LIN {X 0,Y 230.991,Z 464.368,A -85,B 0,C 180,E1 -21092.538,E2 -21092.538} C_VEL
LIN {X 0,Y 229.288,Z 474.072,A -85,B 0,C 180,E1 -21093.412,E2 -21093.412} C_VEL
LIN {X 0,Y 227.158,Z 483.891,A -85,B 0,C 180,E1 -21094.538,E2 -21094.538} C_VEL
LIN {X 0,Y 224.562,Z 493.981,A -85,B 0,C 180,E1 -21096.008,E2 -21096.008} C_VEL
LIN {X 0,Y 221.905,Z 503.043,A -85,B 0,C 180,E1 -21097.648,E2 -21097.648} C_VEL
LIN {X 0,Y 218.983,Z 511.866,A -85,B 0,C 180,E1 -21099.624,E2 -21099.624} C_VEL
LIN {X 0,Y 216.287,Z 519.229,A -85,B 0,C 180,E1 -21101.638,E2 -21101.638} C_VEL
LIN {X 0,Y 213.888,Z 525.476,A -85,B 0,C 180,E1 -21103.707,E2 -21103.707} C_VEL
LIN {X 0,Y 211.783,Z 530.779,A -85,B 0,C 180,E1 -21105.823,E2 -21105.823} C_VEL
LIN {X 0,Y 209.103,Z 537.073,A -85,B 0,C 180,E1 -21109.05,E2 -21109.05} C_VEL
LIN {X 0,Y 207.83,Z 540.216,A -85,B 0,C 180,E1 -21111.057,E2 -21111.057} C_VEL
LIN {X 0,Y 205.854,Z 544.744,A -85,B 0,C 180,E1 -21115.023,E2 -21115.023} C_VEL
LIN {X 0,Y 205.221,Z 546.173,A -85,B 0,C 180,E1 -21116.775,E2 -21116.775} C_VEL
LIN {X 0,Y 204.564,Z 547.552,A -85,B 0,C 180,E1 -21119.194,E2 -21119.194} C_VEL
LIN {X 0,Y 204.178,Z 548.312,A -85,B 0,C 180,E1 -21121.191,E2 -21121.191} C_VEL
LIN {X 0,Y 203.917,Z 548.681,A -85,B 0,C 180,E1 -21123.65,E2 -21123.65} C_VEL
LIN {X 0,Y 203.84,Z 547.791,A -85,B 0,C 180,E1 -21127.712,E2 -21127.712} C_VEL
LIN {X 0,Y 204.07,Z 546.726,A -85,B 0,C 180,E1 -21129.855,E2 -21129.855} C_VEL
LIN {X 0,Y 204.801,Z 543.17,A -85,B 0,C 180,E1 -21133.917,E2 -21133.917} C_VEL
LIN {X 0,Y 205.395,Z 540.506,A -85,B 0,C 180,E1 -21136.142,E2 -21136.142} C_VEL
LIN {X 0,Y 206.522,Z 535.454,A -85,B 0,C 180,E1 -21139.312,E2 -21139.312} C_VEL
LIN {X 0,Y 208.013,Z 529.409,A -85,B 0,C 180,E1 -21142.233,E2 -21142.233} C_VEL
LIN {X 0,Y 209.693,Z 523.042,A -85,B 0,C 180,E1 -21144.712,E2 -21144.712} C_VEL
LIN {X 0,Y 211.428,Z 516.481,A -85,B 0,C 180,E1 -21146.829,E2 -21146.829} C_VEL
LIN {X 0,Y 213.706,Z 506.97,A -85,B 0,C 180,E1 -21149.294,E2 -21149.294} C_VEL
LIN {X 0,Y 215.821,Z 498.001,A -85,B 0,C 180,E1 -21151.166,E2 -21151.166} C_VEL
LIN {X 0,Y 217.545,Z 489.788,A -85,B 0,C 180,E1 -21152.594,E2 -21152.594} C_VEL
LIN {X 0,Y 219.548,Z 478.688,A -85,B 0,C 180,E1 -21154.131,E2 -21154.131} C_VEL
LIN {X 0,Y 221.149,Z 468.369,A -85,B 0,C 180,E1 -21155.242,E2 -21155.242} C_VEL
LIN {X 0,Y 222.36,Z 457.762,A -85,B 0,C 180,E1 -21156.124,E2 -21156.124} C_VEL
LIN {X 0,Y 223.449,Z 446.329,A -85,B 0,C 180,E1 -21156.774,E2 -21156.774} C_VEL
LIN {X 0,Y 224.548,Z 426.084,A -85,B 0,C 180,E1 -21157.478,E2 -21157.478} C_VEL
LIN {X 0,Y 226.379,Z 382.607,A -85,B 0,C 180,E1 -21158.855,E2 -21158.855} C_VEL
LIN {X 0,Y 221.699,Z 370.258,A -85,B 0,C 180,E1 -21159.987,E2 -21159.987} C_VEL
LIN {X 0,Y 215.137,Z 354.309,A -85,B 0,C 180,E1 -21161.622,E2 -21161.622} C_VEL
LIN {X 0,Y 208.262,Z 340.607,A -85,B 0,C 180,E1 -21163.351,E2 -21163.351} C_VEL
LIN {X 0,Y 207.018,Z 337.894,A -85,B 0,C 180,E1 -21163.81,E2 -21163.81} C_VEL
LIN {X 0,Y 206.912,Z 337.294,A -85,B 0,C 180,E1 -21164.256,E2 -21164.256} C_VEL
LIN {X 0,Y 206.86,Z 337.211,A -85,B 0,C 180,E1 -21167.956,E2 -21167.956} C_VEL
LIN {X 0,Y 206.756,Z 337.217,A -85,B 0,C 180,E1 -21173.396,E2 -21173.396} C_VEL
LIN {X 0,Y 206.739,Z 337.215,A -85,B 0,C 180,E1 -21178.42,E2 -21178.42} C_VEL
LIN {X 0,Y 206.708,Z 337.221,A -85,B 0,C 180,E1 -21182.956,E2 -21182.956} C_VEL
LIN {X 0,Y 206.724,Z 337.215,A -85,B 0,C 180,E1 -21185.32,E2 -21185.32} C_VEL
LIN {X 0,Y 206.669,Z 337.222,A -85,B 0,C 180,E1 -21190.25,E2 -21190.25} C_VEL
LIN {X 0,Y 206.637,Z 337.245,A -85,B 0,C 180,E1 -21195.581,E2 -21195.581} C_VEL
LIN {X 0,Y 206.663,Z 337.207,A -85,B 0,C 180,E1 -21199.749,E2 -21199.749} C_VEL
LIN {X 0,Y 206.701,Z 337.234,A -85,B 0,C 180,E1 -21204.689,E2 -21204.689} C_VEL
LIN {X 0,Y 206.697,Z 337.198,A -85,B 0,C 180,E1 -21209.334,E2 -21209.334} C_VEL
LIN {X 0,Y 206.709,Z 337.222,A -85,B 0,C 180,E1 -21213.768,E2 -21213.768} C_VEL
LIN {X 0,Y 206.737,Z 337.222,A -85,B 0,C 180,E1 -21218.04,E2 -21218.04} C_VEL
LIN {X 0,Y 206.828,Z 337.17,A -85,B 0,C 180,E1 -21222.192,E2 -21222.192} C_VEL
LIN {X 0,Y 206.884,Z 337.209,A -85,B 0,C 180,E1 -21226.243,E2 -21226.243} C_VEL
LIN {X 0,Y 207.08,Z 337.176,A -85,B 0,C 180,E1 -21230.23,E2 -21230.23} C_VEL
LIN {X 0,Y 207.04,Z 337.145,A -85,B 0,C 180,E1 -21234.155,E2 -21234.155} C_VEL
LIN {X 0,Y 207.347,Z 337.149,A -85,B 0,C 180,E1 -21238.057,E2 -21238.057} C_VEL
LIN {X 0,Y 207.484,Z 337.138,A -85,B 0,C 180,E1 -21240,E2 -21240} C_VEL
LIN {X 0,Y 207.348,Z 337.138,A -85,B 0,C 180,E1 -21241.942,E2 -21241.942} C_VEL
LIN {X 0,Y 207.134,Z 337.166,A -85,B 0,C 180,E1 -21247.8,E2 -21247.8} C_VEL
LIN {X 0,Y 207.063,Z 337.192,A -85,B 0,C 180,E1 -21250.164,E2 -21250.164} C_VEL
LIN {X 0,Y 206.801,Z 337.189,A -85,B 0,C 180,E1 -21255.775,E2 -21255.775} C_VEL
LIN {X 0,Y 206.714,Z 337.237,A -85,B 0,C 180,E1 -21259.875,E2 -21259.875} C_VEL
LIN {X 0,Y 206.735,Z 337.204,A -85,B 0,C 180,E1 -21264.075,E2 -21264.075} C_VEL
LIN {X 0,Y 206.689,Z 337.238,A -85,B 0,C 180,E1 -21268.426,E2 -21268.426} C_VEL
LIN {X 0,Y 206.694,Z 337.228,A -85,B 0,C 180,E1 -21272.958,E2 -21272.958} C_VEL
LIN {X 0,Y 206.699,Z 337.235,A -85,B 0,C 180,E1 -21275.311,E2 -21275.311} C_VEL
LIN {X 0,Y 206.643,Z 337.245,A -85,B 0,C 180,E1 -21280.255,E2 -21280.255} C_VEL
LIN {X 0,Y 206.622,Z 337.243,A -85,B 0,C 180,E1 -21285.355,E2 -21285.355} C_VEL
LIN {X 0,Y 206.702,Z 337.357,A -85,B 0,C 180,E1 -21289.626,E2 -21289.626} C_VEL
LIN {X 0,Y 207.203,Z 339.383,A -85,B 0,C 180,E1 -21290.808,E2 -21290.808} C_VEL
LIN {X 0,Y 207.694,Z 341.656,A -85,B 0,C 180,E1 -21291.645,E2 -21291.645} C_VEL
LIN {X 0,Y 208.362,Z 345.527,A -85,B 0,C 180,E1 -21292.422,E2 -21292.422} C_VEL
LIN {X 0,Y 209.256,Z 351.887,A -85,B 0,C 180,E1 -21293.126,E2 -21293.126} C_VEL
LIN {X 0,Y 211.154,Z 364.004,A -85,B 0,C 180,E1 -21293.947,E2 -21293.947} C_VEL
LIN {X 0,Y 212.237,Z 367.853,A -85,B 0,C 180,E1 -21294.286,E2 -21294.286} C_VEL
LIN {X 0,Y 218.175,Z 383.461,A -85,B 0,C 180,E1 -21295.828,E2 -21295.828} C_VEL
LIN {X 0,Y 219.745,Z 395.439,A -85,B 0,C 180,E1 -21296.523,E2 -21296.523} C_VEL
LIN {X 0,Y 217.151,Z 449.684,A -85,B 0,C 180,E1 -21298.324,E2 -21298.324} C_VEL
LIN {X 0,Y 216.405,Z 459.263,A -85,B 0,C 180,E1 -21298.829,E2 -21298.829} C_VEL
LIN {X 0,Y 215.141,Z 469.584,A -85,B 0,C 180,E1 -21299.579,E2 -21299.579} C_VEL
LIN {X 0,Y 213.699,Z 478.713,A -85,B 0,C 180,E1 -21300.441,E2 -21300.441} C_VEL
LIN {X 0,Y 211.865,Z 489.444,A -85,B 0,C 180,E1 -21301.79,E2 -21301.79} C_VEL
LIN {X 0,Y 209.66,Z 499.462,A -85,B 0,C 180,E1 -21303.362,E2 -21303.362} C_VEL
LIN {X 0,Y 207.477,Z 508.858,A -85,B 0,C 180,E1 -21305.217,E2 -21305.217} C_VEL
LIN {X 0,Y 205.84,Z 515.883,A -85,B 0,C 180,E1 -21306.881,E2 -21306.881} C_VEL
LIN {X 0,Y 203.685,Z 524.444,A -85,B 0,C 180,E1 -21309.374,E2 -21309.374} C_VEL
LIN {X 0,Y 201.845,Z 531.126,A -85,B 0,C 180,E1 -21311.737,E2 -21311.737} C_VEL
LIN {X 0,Y 200.242,Z 536.899,A -85,B 0,C 180,E1 -21314.216,E2 -21314.216} C_VEL
LIN {X 0,Y 199.057,Z 541.697,A -85,B 0,C 180,E1 -21316.733,E2 -21316.733} C_VEL
LIN {X 0,Y 198.081,Z 546.272,A -85,B 0,C 180,E1 -21319.781,E2 -21319.781} C_VEL
LIN {X 0,Y 197.345,Z 550.566,A -85,B 0,C 180,E1 -21323.867,E2 -21323.867} C_VEL
LIN {X 0,Y 197.144,Z 552.501,A -85,B 0,C 180,E1 -21326.525,E2 -21326.525} C_VEL
LIN {X 0,Y 197.242,Z 553.89,A -85,B 0,C 180,E1 -21330,E2 -21330} C_VEL
LIN {X 0,Y 197.19,Z 554.197,A -85,B 0,C 180,E1 -21332.042,E2 -21332.042} C_VEL
LIN {X 0,Y 197.408,Z 553.575,A -85,B 0,C 180,E1 -21336.131,E2 -21336.131} C_VEL
LIN {X 0,Y 198.182,Z 551.263,A -85,B 0,C 180,E1 -21340.213,E2 -21340.213} C_VEL
LIN {X 0,Y 199.305,Z 548.5,A -85,B 0,C 180,E1 -21343.25,E2 -21343.25} C_VEL
LIN {X 0,Y 200.827,Z 544.728,A -85,B 0,C 180,E1 -21346.258,E2 -21346.258} C_VEL
LIN {X 0,Y 203.105,Z 539.836,A -85,B 0,C 180,E1 -21349.191,E2 -21349.191} C_VEL
LIN {X 0,Y 205.282,Z 534.853,A -85,B 0,C 180,E1 -21351.594,E2 -21351.594} C_VEL
LIN {X 0,Y 208.16,Z 527.463,A -85,B 0,C 180,E1 -21354.43,E2 -21354.43} C_VEL
LIN {X 0,Y 211.104,Z 519.997,A -85,B 0,C 180,E1 -21356.707,E2 -21356.707} C_VEL
LIN {X 0,Y 213.733,Z 512.974,A -85,B 0,C 180,E1 -21358.476,E2 -21358.476} C_VEL
LIN {X 0,Y 216.843,Z 503.458,A -85,B 0,C 180,E1 -21360.425,E2 -21360.425} C_VEL
LIN {X 0,Y 219.6,Z 494.547,A -85,B 0,C 180,E1 -21361.874,E2 -21361.874} C_VEL
LIN {X 0,Y 221.939,Z 485.384,A -85,B 0,C 180,E1 -21363.11,E2 -21363.11} C_VEL
LIN {X 0,Y 224.415,Z 473.711,A -85,B 0,C 180,E1 -21364.312,E2 -21364.312} C_VEL
LIN {X 0,Y 226.285,Z 462.828,A -85,B 0,C 180,E1 -21365.138,E2 -21365.138} C_VEL
LIN {X 0,Y 227.665,Z 452.178,A -85,B 0,C 180,E1 -21365.706,E2 -21365.706} C_VEL
LIN {X 0,Y 228.836,Z 433.635,A -85,B 0,C 180,E1 -21366.376,E2 -21366.376} C_VEL
LIN {X 0,Y 230.861,Z 397.556,A -85,B 0,C 180,E1 -21367.506,E2 -21367.506} C_VEL
LIN {X 0,Y 230.289,Z 394.728,A -85,B 0,C 180,E1 -21367.764,E2 -21367.764} C_VEL
LIN {X 0,Y 225.862,Z 383.934,A -85,B 0,C 180,E1 -21369.337,E2 -21369.337} C_VEL
LIN {X 0,Y 221.04,Z 373.739,A -85,B 0,C 180,E1 -21371.113,E2 -21371.113} C_VEL
LIN {X 0,Y 215.575,Z 363.857,A -85,B 0,C 180,E1 -21373.241,E2 -21373.241} C_VEL
LIN {X 0,Y 211.072,Z 356.624,A -85,B 0,C 180,E1 -21375.117,E2 -21375.117} C_VEL
LIN {X 0,Y 207.674,Z 351.407,A -85,B 0,C 180,E1 -21376.652,E2 -21376.652} C_VEL
LIN {X 0,Y 203.916,Z 345.962,A -85,B 0,C 180,E1 -21378.495,E2 -21378.495} C_VEL
LIN {X 0,Y 200.8,Z 341.569,A -85,B 0,C 180,E1 -21380.188,E2 -21380.188} C_VEL
LIN {X 0,Y 200.327,Z 340.412,A -85,B 0,C 180,E1 -21380.841,E2 -21380.841} C_VEL
LIN {X 0,Y 199.603,Z 338.146,A -85,B 0,C 180,E1 -21383.076,E2 -21383.076} C_VEL
LIN {X 0,Y 199.693,Z 338.1,A -85,B 0,C 180,E1 -21388.136,E2 -21388.136} C_VEL
LIN {X 0,Y 199.686,Z 338.099,A -85,B 0,C 180,E1 -21392.772,E2 -21392.772} C_VEL
LIN {X 0,Y 199.738,Z 338.091,A -85,B 0,C 180,E1 -21397.23,E2 -21397.23} C_VEL
LIN {X 0,Y 199.797,Z 338.082,A -85,B 0,C 180,E1 -21401.758,E2 -21401.758} C_VEL
LIN {X 0,Y 199.849,Z 338.076,A -85,B 0,C 180,E1 -21405.75,E2 -21405.75} C_VEL
LIN {X 0,Y 200.076,Z 338.052,A -85,B 0,C 180,E1 -21409.885,E2 -21409.885} C_VEL
LIN {X 0,Y 200.039,Z 338.065,A -85,B 0,C 180,E1 -21413.95,E2 -21413.95} C_VEL
LIN {X 0,Y 200.324,Z 338.032,A -85,B 0,C 180,E1 -21417.99,E2 -21417.99} C_VEL
LIN {X 0,Y 200.481,Z 337.999,A -85,B 0,C 180,E1 -21420,E2 -21420} C_VEL
LIN {X 0,Y 200.034,Z 338.057,A -85,B 0,C 180,E1 -21424.03,E2 -21424.03} C_VEL
LIN {X 0,Y 200.134,Z 338.047,A -85,B 0,C 180,E1 -21428.075,E2 -21428.075} C_VEL
LIN {X 0,Y 199.889,Z 338.077,A -85,B 0,C 180,E1 -21432.179,E2 -21432.179} C_VEL
LIN {X 0,Y 199.833,Z 338.258,A -85,B 0,C 180,E1 -21435.36,E2 -21435.36} C_VEL
LIN {X 0,Y 201.002,Z 341.243,A -85,B 0,C 180,E1 -21436.179,E2 -21436.179} C_VEL
LIN {X 0,Y 203.144,Z 343.29,A -85,B 0,C 180,E1 -21437.253,E2 -21437.253} C_VEL
LIN {X 0,Y 203.866,Z 343.978,A -85,B 0,C 180,E1 -21437.603,E2 -21437.603} C_VEL
LIN {X 0,Y 205.814,Z 347.16,A -85,B 0,C 180,E1 -21438.607,E2 -21438.607} C_VEL
LIN {X 0,Y 207.679,Z 349.151,A -85,B 0,C 180,E1 -21439.459,E2 -21439.459} C_VEL
LIN {X 0,Y 211.882,Z 355.373,A -85,B 0,C 180,E1 -21441.336,E2 -21441.336} C_VEL
LIN {X 0,Y 216.905,Z 363.24,A -85,B 0,C 180,E1 -21443.386,E2 -21443.386} C_VEL
LIN {X 0,Y 223.704,Z 375.723,A -85,B 0,C 180,E1 -21445.955,E2 -21445.955} C_VEL
LIN {X 0,Y 228.725,Z 386.551,A -85,B 0,C 180,E1 -21447.746,E2 -21447.746} C_VEL
LIN {X 0,Y 231.231,Z 393.178,A -85,B 0,C 180,E1 -21448.632,E2 -21448.632} C_VEL
LIN {X 0,Y 228.008,Z 444.485,A -85,B 0,C 180,E1 -21450.237,E2 -21450.237} C_VEL
LIN {X 0,Y 226.966,Z 454.3,A -85,B 0,C 180,E1 -21450.71,E2 -21450.71} C_VEL
LIN {X 0,Y 225.472,Z 464.664,A -85,B 0,C 180,E1 -21451.429,E2 -21451.429} C_VEL
LIN {X 0,Y 223.773,Z 473.933,A -85,B 0,C 180,E1 -21452.271,E2 -21452.271} C_VEL
LIN {X 0,Y 221.315,Z 484.658,A -85,B 0,C 180,E1 -21453.531,E2 -21453.531} C_VEL
LIN {X 0,Y 218.917,Z 493.605,A -85,B 0,C 180,E1 -21454.849,E2 -21454.849} C_VEL
LIN {X 0,Y 215.848,Z 503.572,A -85,B 0,C 180,E1 -21456.699,E2 -21456.699} C_VEL
LIN {X 0,Y 213.037,Z 511.63,A -85,B 0,C 180,E1 -21458.535,E2 -21458.535} C_VEL
LIN {X 0,Y 210.307,Z 518.789,A -85,B 0,C 180,E1 -21460.514,E2 -21460.514} C_VEL
LIN {X 0,Y 207.111,Z 526.53,A -85,B 0,C 180,E1 -21463.194,E2 -21463.194} C_VEL
LIN {X 0,Y 204.962,Z 531.617,A -85,B 0,C 180,E1 -21465.339,E2 -21465.339} C_VEL
LIN {X 0,Y 203.064,Z 535.949,A -85,B 0,C 180,E1 -21467.555,E2 -21467.555} C_VEL
LIN {X 0,Y 200.741,Z 541.076,A -85,B 0,C 180,E1 -21470.936,E2 -21470.936} C_VEL
LIN {X 0,Y 198.994,Z 544.736,A -85,B 0,C 180,E1 -21474.322,E2 -21474.322} C_VEL
LIN {X 0,Y 197.585,Z 547.577,A -85,B 0,C 180,E1 -21478.614,E2 -21478.614} C_VEL
LIN {X 0,Y 197.275,Z 548.247,A -85,B 0,C 180,E1 -21480.083,E2 -21480.083} C_VEL
LIN {X 0,Y 196.838,Z 548.764,A -85,B 0,C 180,E1 -21483.204,E2 -21483.204} C_VEL
LIN {X 0,Y 196.711,Z 548.233,A -85,B 0,C 180,E1 -21486.859,E2 -21486.859} C_VEL
LIN {X 0,Y 196.862,Z 547.189,A -85,B 0,C 180,E1 -21489.084,E2 -21489.084} C_VEL
LIN {X 0,Y 197.159,Z 545.745,A -85,B 0,C 180,E1 -21491.288,E2 -21491.288} C_VEL
LIN {X 0,Y 197.656,Z 543.611,A -85,B 0,C 180,E1 -21493.747,E2 -21493.747} C_VEL
LIN {X 0,Y 198.437,Z 540.125,A -85,B 0,C 180,E1 -21496.691,E2 -21496.691} C_VEL
LIN {X 0,Y 199.753,Z 534.627,A -85,B 0,C 180,E1 -21500.111,E2 -21500.111} C_VEL
LIN {X 0,Y 201.304,Z 528.712,A -85,B 0,C 180,E1 -21502.981,E2 -21502.981} C_VEL
LIN {X 0,Y 203.073,Z 522.187,A -85,B 0,C 180,E1 -21505.534,E2 -21505.534} C_VEL
LIN {X 0,Y 205.192,Z 514.275,A -85,B 0,C 180,E1 -21508.037,E2 -21508.037} C_VEL
LIN {X 0,Y 207.068,Z 506.764,A -85,B 0,C 180,E1 -21510,E2 -21510} C_VEL
LIN {X 0,Y 209.299,Z 497.72,A -85,B 0,C 180,E1 -21511.924,E2 -21511.924} C_VEL
LIN {X 0,Y 211.234,Z 488.729,A -85,B 0,C 180,E1 -21513.494,E2 -21513.494} C_VEL
LIN {X 0,Y 212.863,Z 480.134,A -85,B 0,C 180,E1 -21514.735,E2 -21514.735} C_VEL
LIN {X 0,Y 214.691,Z 468.951,A -85,B 0,C 180,E1 -21515.99,E2 -21515.99} C_VEL
LIN {X 0,Y 215.997,Z 457.719,A -85,B 0,C 180,E1 -21516.95,E2 -21516.95} C_VEL
LIN {X 0,Y 217.092,Z 447.007,A -85,B 0,C 180,E1 -21517.578,E2 -21517.578} C_VEL
LIN {X 0,Y 218.099,Z 429.281,A -85,B 0,C 180,E1 -21518.229,E2 -21518.229} C_VEL
LIN {X 0,Y 220.105,Z 384.246,A -85,B 0,C 180,E1 -21519.686,E2 -21519.686} C_VEL
LIN {X 0,Y 215.374,Z 371.866,A -85,B 0,C 180,E1 -21520.883,E2 -21520.883} C_VEL
LIN {X 0,Y 209.688,Z 357.873,A -85,B 0,C 180,E1 -21522.375,E2 -21522.375} C_VEL
LIN {X 0,Y 202.814,Z 344.277,A -85,B 0,C 180,E1 -21524.162,E2 -21524.162} C_VEL
LIN {X 0,Y 200.134,Z 339.336,A -85,B 0,C 180,E1 -21524.912,E2 -21524.912} C_VEL
LIN {X 0,Y 199.868,Z 338.298,A -85,B 0,C 180,E1 -21525.29,E2 -21525.29} C_VEL
LIN {X 0,Y 199.783,Z 338.09,A -85,B 0,C 180,E1 -21528.458,E2 -21528.458} C_VEL
LIN {X 0,Y 199.717,Z 338.095,A -85,B 0,C 180,E1 -21533.803,E2 -21533.803} C_VEL
LIN {X 0,Y 199.71,Z 338.09,A -85,B 0,C 180,E1 -21538.384,E2 -21538.384} C_VEL
LIN {X 0,Y 199.66,Z 338.107,A -85,B 0,C 180,E1 -21542.349,E2 -21542.349} C_VEL
LIN {X 0,Y 199.642,Z 338.113,A -85,B 0,C 180,E1 -21546.759,E2 -21546.759} C_VEL
LIN {X 0,Y 199.641,Z 338.108,A -85,B 0,C 180,E1 -21549.321,E2 -21549.321} C_VEL
LIN {X 0,Y 199.584,Z 338.12,A -85,B 0,C 180,E1 -21554.77,E2 -21554.77} C_VEL
LIN {X 0,Y 199.582,Z 338.107,A -85,B 0,C 180,E1 -21558.005,E2 -21558.005} C_VEL
LIN {X 0,Y 199.612,Z 338.082,A -85,B 0,C 180,E1 -21560.768,E2 -21560.768} C_VEL
LIN {X 0,Y 199.613,Z 338.119,A -85,B 0,C 180,E1 -21565.713,E2 -21565.713} C_VEL
LIN {X 0,Y 199.688,Z 338.087,A -85,B 0,C 180,E1 -21568.134,E2 -21568.134} C_VEL
LIN {X 0,Y 199.646,Z 338.086,A -85,B 0,C 180,E1 -21572.765,E2 -21572.765} C_VEL
LIN {X 0,Y 199.711,Z 338.104,A -85,B 0,C 180,E1 -21577.225,E2 -21577.225} C_VEL
LIN {X 0,Y 199.752,Z 338.05,A -85,B 0,C 180,E1 -21581.798,E2 -21581.798} C_VEL
LIN {X 0,Y 199.821,Z 338.082,A -85,B 0,C 180,E1 -21585.747,E2 -21585.747} C_VEL
LIN {X 0,Y 200.025,Z 338.056,A -85,B 0,C 180,E1 -21589.881,E2 -21589.881} C_VEL
LIN {X 0,Y 200.004,Z 338.02,A -85,B 0,C 180,E1 -21593.948,E2 -21593.948} C_VEL
LIN {X 0,Y 200.289,Z 338.028,A -85,B 0,C 180,E1 -21597.989,E2 -21597.989} C_VEL
LIN {X 0,Y 200.451,Z 338.014,A -85,B 0,C 180,E1 -21600,E2 -21600} C_VEL
LIN {X 0,Y 199.993,Z 338.029,A -85,B 0,C 180,E1 -21604.03,E2 -21604.03} C_VEL
LIN {X 0,Y 200.084,Z 338.048,A -85,B 0,C 180,E1 -21608.076,E2 -21608.076} C_VEL
LIN {X 0,Y 199.857,Z 338.08,A -85,B 0,C 180,E1 -21612.18,E2 -21612.18} C_VEL
LIN {X 0,Y 199.742,Z 338.072,A -85,B 0,C 180,E1 -21616.348,E2 -21616.348} C_VEL
LIN {X 0,Y 199.647,Z 338.113,A -85,B 0,C 180,E1 -21620.61,E2 -21620.61} C_VEL
LIN {X 0,Y 199.649,Z 338.09,A -85,B 0,C 180,E1 -21624.987,E2 -21624.987} C_VEL
LIN {X 0,Y 199.609,Z 338.109,A -85,B 0,C 180,E1 -21629.532,E2 -21629.532} C_VEL
LIN {X 0,Y 199.665,Z 338.096,A -85,B 0,C 180,E1 -21632.352,E2 -21632.352} C_VEL
LIN {X 0,Y 199.614,Z 338.104,A -85,B 0,C 180,E1 -21636.764,E2 -21636.764} C_VEL
LIN {X 0,Y 199.592,Z 338.12,A -85,B 0,C 180,E1 -21639.331,E2 -21639.331} C_VEL
LIN {X 0,Y 199.563,Z 338.113,A -85,B 0,C 180,E1 -21642.306,E2 -21642.306} C_VEL
LIN {X 0,Y 199.575,Z 338.123,A -85,B 0,C 180,E1 -21645.227,E2 -21645.227} C_VEL
LIN {X 0,Y 199.654,Z 338.34,A -85,B 0,C 180,E1 -21648.805,E2 -21648.805} C_VEL
LIN {X 0,Y 200.775,Z 342.66,A -85,B 0,C 180,E1 -21651.153,E2 -21651.153} C_VEL
LIN {X 0,Y 206.804,Z 355.302,A -85,B 0,C 180,E1 -21652.852,E2 -21652.852} C_VEL
LIN {X 0,Y 212.237,Z 367.853,A -85,B 0,C 180,E1 -21654.286,E2 -21654.286} C_VEL
LIN {X 0,Y 213.639,Z 373.386,A -85,B 0,C 180,E1 -21654.735,E2 -21654.735} C_VEL
LIN {X 0,Y 214.2,Z 379.209,A -85,B 0,C 180,E1 -21655.058,E2 -21655.058} C_VEL
LIN {X 0,Y 213.825,Z 391.21,A -85,B 0,C 180,E1 -21655.485,E2 -21655.485} C_VEL
LIN {X 0,Y 213.327,Z 399.271,A -85,B 0,C 180,E1 -21655.734,E2 -21655.734} C_VEL
LIN {X 0,Y 210.886,Z 449.057,A -85,B 0,C 180,E1 -21657.431,E2 -21657.431} C_VEL
LIN {X 0,Y 210.138,Z 458.563,A -85,B 0,C 180,E1 -21657.931,E2 -21657.931} C_VEL
LIN {X 0,Y 208.851,Z 469.048,A -85,B 0,C 180,E1 -21658.702,E2 -21658.702} C_VEL
LIN {X 0,Y 207.18,Z 479.208,A -85,B 0,C 180,E1 -21659.695,E2 -21659.695} C_VEL
LIN {X 0,Y 205.275,Z 489.825,A -85,B 0,C 180,E1 -21661.079,E2 -21661.079} C_VEL
LIN {X 0,Y 202.989,Z 499.756,A -85,B 0,C 180,E1 -21662.693,E2 -21662.693} C_VEL
LIN {X 0,Y 201.004,Z 508.057,A -85,B 0,C 180,E1 -21664.362,E2 -21664.362} C_VEL
LIN {X 0,Y 198.806,Z 516.925,A -85,B 0,C 180,E1 -21666.565,E2 -21666.565} C_VEL
LIN {X 0,Y 196.947,Z 524.021,A -85,B 0,C 180,E1 -21668.695,E2 -21668.695} C_VEL
LIN {X 0,Y 195.046,Z 530.628,A -85,B 0,C 180,E1 -21671.077,E2 -21671.077} C_VEL
LIN {X 0,Y 193.081,Z 537.444,A -85,B 0,C 180,E1 -21674.157,E2 -21674.157} C_VEL
LIN {X 0,Y 191.715,Z 542.899,A -85,B 0,C 180,E1 -21677.294,E2 -21677.294} C_VEL
LIN {X 0,Y 191.07,Z 545.952,A -85,B 0,C 180,E1 -21679.402,E2 -21679.402} C_VEL
LIN {X 0,Y 190.424,Z 549.47,A -85,B 0,C 180,E1 -21682.578,E2 -21682.578} C_VEL
LIN {X 0,Y 190.087,Z 551.956,A -85,B 0,C 180,E1 -21685.759,E2 -21685.759} C_VEL
LIN {X 0,Y 190.15,Z 553.763,A -85,B 0,C 180,E1 -21690,E2 -21690} C_VEL
LIN {X 0,Y 190.092,Z 554.066,A -85,B 0,C 180,E1 -21693.418,E2 -21693.418} C_VEL
LIN {X 0,Y 190.352,Z 553.546,A -85,B 0,C 180,E1 -21696.359,E2 -21696.359} C_VEL
LIN {X 0,Y 191.17,Z 551.297,A -85,B 0,C 180,E1 -21700.592,E2 -21700.592} C_VEL
LIN {X 0,Y 192.375,Z 548.591,A -85,B 0,C 180,E1 -21703.737,E2 -21703.737} C_VEL
LIN {X 0,Y 194.008,Z 544.878,A -85,B 0,C 180,E1 -21706.846,E2 -21706.846} C_VEL
LIN {X 0,Y 196.412,Z 540.061,A -85,B 0,C 180,E1 -21709.872,E2 -21709.872} C_VEL
LIN {X 0,Y 198.689,Z 535.165,A -85,B 0,C 180,E1 -21712.349,E2 -21712.349} C_VEL
LIN {X 0,Y 201.727,Z 527.881,A -85,B 0,C 180,E1 -21715.263,E2 -21715.263} C_VEL
LIN {X 0,Y 204.818,Z 520.519,A -85,B 0,C 180,E1 -21717.596,E2 -21717.596} C_VEL
LIN {X 0,Y 207.895,Z 512.607,A -85,B 0,C 180,E1 -21719.63,E2 -21719.63} C_VEL
LIN {X 0,Y 211.209,Z 503.03,A -85,B 0,C 180,E1 -21721.606,E2 -21721.606} C_VEL
LIN {X 0,Y 214.065,Z 494.05,A -85,B 0,C 180,E1 -21723.08,E2 -21723.08} C_VEL
LIN {X 0,Y 216.521,Z 484.788,A -85,B 0,C 180,E1 -21724.331,E2 -21724.331} C_VEL
LIN {X 0,Y 218.881,Z 474.157,A -85,B 0,C 180,E1 -21725.448,E2 -21725.448} C_VEL
LIN {X 0,Y 220.931,Z 462.669,A -85,B 0,C 180,E1 -21726.333,E2 -21726.333} C_VEL
LIN {X 0,Y 222.353,Z 452.001,A -85,B 0,C 180,E1 -21726.908,E2 -21726.908} C_VEL
LIN {X 0,Y 223.571,Z 433.989,A -85,B 0,C 180,E1 -21727.57,E2 -21727.57} C_VEL
LIN {X 0,Y 225.662,Z 398.776,A -85,B 0,C 180,E1 -21728.691,E2 -21728.691} C_VEL
LIN {X 0,Y 221.567,Z 388.303,A -85,B 0,C 180,E1 -21730.249,E2 -21730.249} C_VEL
LIN {X 0,Y 216.908,Z 378.241,A -85,B 0,C 180,E1 -21732.067,E2 -21732.067} C_VEL
LIN {X 0,Y 211.283,Z 367.762,A -85,B 0,C 180,E1 -21734.412,E2 -21734.412} C_VEL
LIN {X 0,Y 204.983,Z 357.55,A -85,B 0,C 180,E1 -21737.301,E2 -21737.301} C_VEL
LIN {X 0,Y 200.852,Z 351.538,A -85,B 0,C 180,E1 -21739.413,E2 -21739.413} C_VEL
LIN {X 0,Y 196.941,Z 346.172,A -85,B 0,C 180,E1 -21741.599,E2 -21741.599} C_VEL
LIN {X 0,Y 193.033,Z 340.765,A -85,B 0,C 180,E1 -21744.244,E2 -21744.244} C_VEL
LIN {X 0,Y 192.572,Z 339.065,A -85,B 0,C 180,E1 -21746.025,E2 -21746.025} C_VEL
LIN {X 0,Y 192.648,Z 338.984,A -85,B 0,C 180,E1 -21751.109,E2 -21751.109} C_VEL
LIN {X 0,Y 192.706,Z 338.968,A -85,B 0,C 180,E1 -21756.349,E2 -21756.349} C_VEL
LIN {X 0,Y 192.732,Z 338.962,A -85,B 0,C 180,E1 -21761.458,E2 -21761.458} C_VEL
LIN {X 0,Y 192.773,Z 338.96,A -85,B 0,C 180,E1 -21765.215,E2 -21765.215} C_VEL
LIN {X 0,Y 193.021,Z 338.934,A -85,B 0,C 180,E1 -21769.511,E2 -21769.511} C_VEL
LIN {X 0,Y 193.003,Z 338.944,A -85,B 0,C 180,E1 -21773.729,E2 -21773.729} C_VEL
LIN {X 0,Y 193.266,Z 338.91,A -85,B 0,C 180,E1 -21777.917,E2 -21777.917} C_VEL
LIN {X 0,Y 193.445,Z 338.875,A -85,B 0,C 180,E1 -21780.001,E2 -21780.001} C_VEL
LIN {X 0,Y 192.981,Z 338.935,A -85,B 0,C 180,E1 -21784.177,E2 -21784.177} C_VEL
LIN {X 0,Y 193.081,Z 338.924,A -85,B 0,C 180,E1 -21788.372,E2 -21788.372} C_VEL
LIN {X 0,Y 192.9,Z 339.125,A -85,B 0,C 180,E1 -21791.893,E2 -21791.893} C_VEL
LIN {X 0,Y 193.757,Z 341.715,A -85,B 0,C 180,E1 -21792.63,E2 -21792.63} C_VEL
LIN {X 0,Y 195.632,Z 343.816,A -85,B 0,C 180,E1 -21793.82,E2 -21793.82} C_VEL
LIN {X 0,Y 197.126,Z 344.902,A -85,B 0,C 180,E1 -21794.65,E2 -21794.65} C_VEL
LIN {X 0,Y 198.873,Z 347.938,A -85,B 0,C 180,E1 -21795.698,E2 -21795.698} C_VEL
LIN {X 0,Y 201.182,Z 350.339,A -85,B 0,C 180,E1 -21796.899,E2 -21796.899} C_VEL
LIN {X 0,Y 203.625,Z 353.786,A -85,B 0,C 180,E1 -21798.163,E2 -21798.163} C_VEL
LIN {X 0,Y 204.977,Z 355.5,A -85,B 0,C 180,E1 -21798.815,E2 -21798.815} C_VEL
LIN {X 0,Y 208.64,Z 361.017,A -85,B 0,C 180,E1 -21800.535,E2 -21800.535} C_VEL
LIN {X 0,Y 213.19,Z 368.292,A -85,B 0,C 180,E1 -21802.492,E2 -21802.492} C_VEL
LIN {X 0,Y 219.634,Z 380.477,A -85,B 0,C 180,E1 -21805.082,E2 -21805.082} C_VEL
LIN {X 0,Y 224.103,Z 390.285,A -85,B 0,C 180,E1 -21806.76,E2 -21806.76} C_VEL
LIN {X 0,Y 225.941,Z 394.893,A -85,B 0,C 180,E1 -21807.444,E2 -21807.444} C_VEL
LIN {X 0,Y 222.727,Z 444.505,A -85,B 0,C 180,E1 -21809.035,E2 -21809.035} C_VEL
LIN {X 0,Y 221.608,Z 454.525,A -85,B 0,C 180,E1 -21809.525,E2 -21809.525} C_VEL
LIN {X 0,Y 220.111,Z 464.484,A -85,B 0,C 180,E1 -21810.221,E2 -21810.221} C_VEL
LIN {X 0,Y 218.19,Z 474.493,A -85,B 0,C 180,E1 -21811.15,E2 -21811.15} C_VEL
LIN {X 0,Y 216.042,Z 483.76,A -85,B 0,C 180,E1 -21812.243,E2 -21812.243} C_VEL
LIN {X 0,Y 213.264,Z 493.557,A -85,B 0,C 180,E1 -21813.685,E2 -21813.685} C_VEL
LIN {X 0,Y 210.267,Z 502.966,A -85,B 0,C 180,E1 -21815.441,E2 -21815.441} C_VEL
LIN {X 0,Y 207.012,Z 511.856,A -85,B 0,C 180,E1 -21817.5,E2 -21817.5} C_VEL
LIN {X 0,Y 203.695,Z 519.999,A -85,B 0,C 180,E1 -21819.854,E2 -21819.854} C_VEL
LIN {X 0,Y 201.062,Z 526.116,A -85,B 0,C 180,E1 -21822.021,E2 -21822.021} C_VEL
LIN {X 0,Y 198.165,Z 532.449,A -85,B 0,C 180,E1 -21824.822,E2 -21824.822} C_VEL
LIN {X 0,Y 196.185,Z 536.692,A -85,B 0,C 180,E1 -21827.106,E2 -21827.106} C_VEL
LIN {X 0,Y 193.758,Z 541.601,A -85,B 0,C 180,E1 -21830.598,E2 -21830.598} C_VEL
LIN {X 0,Y 191.931,Z 545.158,A -85,B 0,C 180,E1 -21834.135,E2 -21834.135} C_VEL
LIN {X 0,Y 191.076,Z 546.927,A -85,B 0,C 180,E1 -21836.515,E2 -21836.515} C_VEL
LIN {X 0,Y 190.419,Z 548.003,A -85,B 0,C 180,E1 -21838.888,E2 -21838.888} C_VEL
LIN {X 0,Y 189.793,Z 548.835,A -85,B 0,C 180,E1 -21842.713,E2 -21842.713} C_VEL
LIN {X 0,Y 189.614,Z 548.487,A -85,B 0,C 180,E1 -21845.939,E2 -21845.939} C_VEL
LIN {X 0,Y 189.705,Z 547.642,A -85,B 0,C 180,E1 -21848.256,E2 -21848.256} C_VEL
LIN {X 0,Y 189.921,Z 546.432,A -85,B 0,C 180,E1 -21850.547,E2 -21850.547} C_VEL
LIN {X 0,Y 190.508,Z 544.021,A -85,B 0,C 180,E1 -21853.571,E2 -21853.571} C_VEL
LIN {X 0,Y 191.518,Z 539.678,A -85,B 0,C 180,E1 -21857.281,E2 -21857.281} C_VEL
LIN {X 0,Y 192.607,Z 535.318,A -85,B 0,C 180,E1 -21860.132,E2 -21860.132} C_VEL
LIN {X 0,Y 194.274,Z 529.208,A -85,B 0,C 180,E1 -21863.248,E2 -21863.248} C_VEL
LIN {X 0,Y 196.105,Z 522.76,A -85,B 0,C 180,E1 -21865.89,E2 -21865.89} C_VEL
LIN {X 0,Y 197.855,Z 516.708,A -85,B 0,C 180,E1 -21867.965,E2 -21867.965} C_VEL
LIN {X 0,Y 200.228,Z 507.539,A -85,B 0,C 180,E1 -21870.503,E2 -21870.503} C_VEL
LIN {X 0,Y 202.524,Z 498.631,A -85,B 0,C 180,E1 -21872.486,E2 -21872.486} C_VEL
LIN {X 0,Y 204.622,Z 489.273,A -85,B 0,C 180,E1 -21874.187,E2 -21874.187} C_VEL
LIN {X 0,Y 206.519,Z 479.537,A -85,B 0,C 180,E1 -21875.615,E2 -21875.615} C_VEL
LIN {X 0,Y 208.239,Z 469.401,A -85,B 0,C 180,E1 -21876.784,E2 -21876.784} C_VEL
LIN {X 0,Y 209.681,Z 457.57,A -85,B 0,C 180,E1 -21877.817,E2 -21877.817} C_VEL
LIN {X 0,Y 210.786,Z 447.073,A -85,B 0,C 180,E1 -21878.445,E2 -21878.445} C_VEL
LIN {X 0,Y 211.956,Z 427.266,A -85,B 0,C 180,E1 -21879.176,E2 -21879.176} C_VEL
LIN {X 0,Y 213.779,Z 385.663,A -85,B 0,C 180,E1 -21880.573,E2 -21880.573} C_VEL
LIN {X 0,Y 205.438,Z 364.227,A -85,B 0,C 180,E1 -21882.833,E2 -21882.833} C_VEL
LIN {X 0,Y 198.62,Z 349.9,A -85,B 0,C 180,E1 -21884.696,E2 -21884.696} C_VEL
LIN {X 0,Y 194.323,Z 342.545,A -85,B 0,C 180,E1 -21885.882,E2 -21885.882} C_VEL
LIN {X 0,Y 192.921,Z 339.813,A -85,B 0,C 180,E1 -21886.399,E2 -21886.399} C_VEL
LIN {X 0,Y 192.761,Z 339.016,A -85,B 0,C 180,E1 -21886.959,E2 -21886.959} C_VEL
LIN {X 0,Y 192.619,Z 338.99,A -85,B 0,C 180,E1 -21891.4,E2 -21891.4} C_VEL
LIN {X 0,Y 192.65,Z 338.977,A -85,B 0,C 180,E1 -21894.213,E2 -21894.213} C_VEL
LIN {X 0,Y 192.646,Z 338.971,A -85,B 0,C 180,E1 -21898.889,E2 -21898.889} C_VEL
LIN {X 0,Y 192.6,Z 338.975,A -85,B 0,C 180,E1 -21903.186,E2 -21903.186} C_VEL
LIN {X 0,Y 192.612,Z 338.986,A -85,B 0,C 180,E1 -21906.607,E2 -21906.607} C_VEL
LIN {X 0,Y 192.526,Z 338.975,A -85,B 0,C 180,E1 -21911.078,E2 -21911.078} C_VEL
LIN {X 0,Y 192.516,Z 339.005,A -85,B 0,C 180,E1 -21916.083,E2 -21916.083} C_VEL
LIN {X 0,Y 192.519,Z 338.966,A -85,B 0,C 180,E1 -21920.051,E2 -21920.051} C_VEL
LIN {X 0,Y 192.563,Z 338.995,A -85,B 0,C 180,E1 -21924.27,E2 -21924.27} C_VEL
LIN {X 0,Y 192.607,Z 338.982,A -85,B 0,C 180,E1 -21927.061,E2 -21927.061} C_VEL
LIN {X 0,Y 192.622,Z 338.947,A -85,B 0,C 180,E1 -21931.685,E2 -21931.685} C_VEL
LIN {X 0,Y 192.682,Z 338.984,A -85,B 0,C 180,E1 -21936.345,E2 -21936.345} C_VEL
LIN {X 0,Y 192.701,Z 338.928,A -85,B 0,C 180,E1 -21941.487,E2 -21941.487} C_VEL
LIN {X 0,Y 192.746,Z 338.957,A -85,B 0,C 180,E1 -21945.212,E2 -21945.212} C_VEL
LIN {X 0,Y 192.947,Z 338.94,A -85,B 0,C 180,E1 -21949.566,E2 -21949.566} C_VEL
LIN {X 0,Y 192.968,Z 338.895,A -85,B 0,C 180,E1 -21953.727,E2 -21953.727} C_VEL
LIN {X 0,Y 193.233,Z 338.906,A -85,B 0,C 180,E1 -21957.915,E2 -21957.915} C_VEL
LIN {X 0,Y 193.417,Z 338.891,A -85,B 0,C 180,E1 -21959.999,E2 -21959.999} C_VEL
LIN {X 0,Y 192.94,Z 338.906,A -85,B 0,C 180,E1 -21964.177,E2 -21964.177} C_VEL
LIN {X 0,Y 193.033,Z 338.93,A -85,B 0,C 180,E1 -21968.373,E2 -21968.373} C_VEL
LIN {X 0,Y 192.778,Z 338.953,A -85,B 0,C 180,E1 -21972.634,E2 -21972.634} C_VEL
LIN {X 0,Y 192.695,Z 338.977,A -85,B 0,C 180,E1 -21978.508,E2 -21978.508} C_VEL
LIN {X 0,Y 192.636,Z 338.959,A -85,B 0,C 180,E1 -21984.204,E2 -21984.204} C_VEL
LIN {X 0,Y 192.602,Z 338.988,A -85,B 0,C 180,E1 -21988.865,E2 -21988.865} C_VEL
LIN {X 0,Y 192.595,Z 338.986,A -85,B 0,C 180,E1 -21993.186,E2 -21993.186} C_VEL
LIN {X 0,Y 192.539,Z 338.987,A -85,B 0,C 180,E1 -21998.354,E2 -21998.354} C_VEL
LIN {X 0,Y 192.482,Z 338.996,A -85,B 0,C 180,E1 -22003.092,E2 -22003.092} C_VEL
LIN {X 0,Y 192.53,Z 339.073,A -85,B 0,C 180,E1 -22007.65,E2 -22007.65} C_VEL
LIN {X 0,Y 193.396,Z 342.363,A -85,B 0,C 180,E1 -22009.641,E2 -22009.641} C_VEL
LIN {X 0,Y 196.185,Z 348.15,A -85,B 0,C 180,E1 -22010.579,E2 -22010.579} C_VEL
LIN {X 0,Y 202.007,Z 360.289,A -85,B 0,C 180,E1 -22012.222,E2 -22012.222} C_VEL
LIN {X 0,Y 209.106,Z 377.488,A -85,B 0,C 180,E1 -22014.176,E2 -22014.176} C_VEL
LIN {X 0,Y 212.256,Z 386.343,A -85,B 0,C 180,E1 -22015.046,E2 -22015.046} C_VEL
LIN {X 0,Y 213.471,Z 396.531,A -85,B 0,C 180,E1 -22015.646,E2 -22015.646} C_VEL
LIN {X 0,Y 213.327,Z 399.271,A -85,B 0,C 180,E1 -22015.734,E2 -22015.734} C_VEL
LIN {X 0,Y 212.506,Z 405.104,A -85,B 0,C 180,E1 -22015.844,E2 -22015.844} C_VEL
LIN {X 0,Y 206.595,Z 424.046,A -85,B 0,C 180,E1 -22015.712,E2 -22015.712} C_VEL
LIN {X 0,Y 205.671,Z 429.883,A -85,B 0,C 180,E1 -22015.811,E2 -22015.811} C_VEL
LIN {X 0,Y 204.527,Z 450.413,A -85,B 0,C 180,E1 -22016.573,E2 -22016.573} C_VEL
LIN {X 0,Y 203.725,Z 459.494,A -85,B 0,C 180,E1 -22017.089,E2 -22017.089} C_VEL
LIN {X 0,Y 202.362,Z 469.692,A -85,B 0,C 180,E1 -22017.873,E2 -22017.873} C_VEL
LIN {X 0,Y 200.698,Z 479.699,A -85,B 0,C 180,E1 -22018.901,E2 -22018.901} C_VEL
LIN {X 0,Y 199.087,Z 488.697,A -85,B 0,C 180,E1 -22020.09,E2 -22020.09} C_VEL
LIN {X 0,Y 196.685,Z 498.808,A -85,B 0,C 180,E1 -22021.741,E2 -22021.741} C_VEL
LIN {X 0,Y 194.3,Z 508.283,A -85,B 0,C 180,E1 -22023.698,E2 -22023.698} C_VEL
LIN {X 0,Y 192.245,Z 516.234,A -85,B 0,C 180,E1 -22025.715,E2 -22025.715} C_VEL
LIN {X 0,Y 190.371,Z 523.171,A -85,B 0,C 180,E1 -22027.819,E2 -22027.819} C_VEL
LIN {X 0,Y 187.966,Z 531.314,A -85,B 0,C 180,E1 -22030.903,E2 -22030.903} C_VEL
LIN {X 0,Y 186.237,Z 537.016,A -85,B 0,C 180,E1 -22033.559,E2 -22033.559} C_VEL
LIN {X 0,Y 184.767,Z 542.539,A -85,B 0,C 180,E1 -22036.807,E2 -22036.807} C_VEL
LIN {X 0,Y 183.783,Z 546.859,A -85,B 0,C 180,E1 -22040.091,E2 -22040.091} C_VEL
LIN {X 0,Y 183.22,Z 550.094,A -85,B 0,C 180,E1 -22043.392,E2 -22043.392} C_VEL
LIN {X 0,Y 182.963,Z 552.501,A -85,B 0,C 180,E1 -22047.082,E2 -22047.082} C_VEL
LIN {X 0,Y 183.06,Z 553.636,A -85,B 0,C 180,E1 -22050,E2 -22050} C_VEL
LIN {X 0,Y 182.985,Z 554.038,A -85,B 0,C 180,E1 -22053.053,E2 -22053.053} C_VEL
LIN {X 0,Y 183.294,Z 553.503,A -85,B 0,C 180,E1 -22056.605,E2 -22056.605} C_VEL
LIN {X 0,Y 184.175,Z 551.337,A -85,B 0,C 180,E1 -22060.999,E2 -22060.999} C_VEL
LIN {X 0,Y 185.465,Z 548.697,A -85,B 0,C 180,E1 -22064.259,E2 -22064.259} C_VEL
LIN {X 0,Y 187.218,Z 545.059,A -85,B 0,C 180,E1 -22067.476,E2 -22067.476} C_VEL
LIN {X 0,Y 189.751,Z 540.315,A -85,B 0,C 180,E1 -22070.601,E2 -22070.601} C_VEL
LIN {X 0,Y 192.575,Z 534.334,A -85,B 0,C 180,E1 -22073.668,E2 -22073.668} C_VEL
LIN {X 0,Y 195.336,Z 528.303,A -85,B 0,C 180,E1 -22076.151,E2 -22076.151} C_VEL
LIN {X 0,Y 198.572,Z 521.043,A -85,B 0,C 180,E1 -22078.542,E2 -22078.542} C_VEL
LIN {X 0,Y 202.165,Z 512.238,A -85,B 0,C 180,E1 -22080.848,E2 -22080.848} C_VEL
LIN {X 0,Y 205.237,Z 503.846,A -85,B 0,C 180,E1 -22082.638,E2 -22082.638} C_VEL
LIN {X 0,Y 208.616,Z 493.614,A -85,B 0,C 180,E1 -22084.353,E2 -22084.353} C_VEL
LIN {X 0,Y 211.192,Z 484.297,A -85,B 0,C 180,E1 -22085.617,E2 -22085.617} C_VEL
LIN {X 0,Y 213.671,Z 473.583,A -85,B 0,C 180,E1 -22086.742,E2 -22086.742} C_VEL
LIN {X 0,Y 215.675,Z 462.77,A -85,B 0,C 180,E1 -22087.587,E2 -22087.587} C_VEL
LIN {X 0,Y 217.149,Z 452.278,A -85,B 0,C 180,E1 -22088.166,E2 -22088.166} C_VEL
LIN {X 0,Y 218.481,Z 433.506,A -85,B 0,C 180,E1 -22088.864,E2 -22088.864} C_VEL
LIN {X 0,Y 220.502,Z 400.822,A -85,B 0,C 180,E1 -22089.922,E2 -22089.922} C_VEL
LIN {X 0,Y 215.883,Z 389.227,A -85,B 0,C 180,E1 -22091.796,E2 -22091.796} C_VEL
LIN {X 0,Y 211.214,Z 379.486,A -85,B 0,C 180,E1 -22093.775,E2 -22093.775} C_VEL
LIN {X 0,Y 206.757,Z 371.358,A -85,B 0,C 180,E1 -22095.776,E2 -22095.776} C_VEL
LIN {X 0,Y 201.874,Z 363.153,A -85,B 0,C 180,E1 -22098.184,E2 -22098.184} C_VEL
LIN {X 0,Y 198.091,Z 357.478,A -85,B 0,C 180,E1 -22100.219,E2 -22100.219} C_VEL
LIN {X 0,Y 194.351,Z 352.169,A -85,B 0,C 180,E1 -22102.438,E2 -22102.438} C_VEL
LIN {X 0,Y 190.085,Z 346.436,A -85,B 0,C 180,E1 -22105.358,E2 -22105.358} C_VEL
LIN {X 0,Y 188.079,Z 344.472,A -85,B 0,C 180,E1 -22106.829,E2 -22106.829} C_VEL
LIN {X 0,Y 186.229,Z 342.18,A -85,B 0,C 180,E1 -22108.346,E2 -22108.346} C_VEL
LIN {X 0,Y 185.643,Z 340.314,A -85,B 0,C 180,E1 -22109.265,E2 -22109.265} C_VEL
LIN {X 0,Y 185.581,Z 339.87,A -85,B 0,C 180,E1 -22110.577,E2 -22110.577} C_VEL
LIN {X 0,Y 185.588,Z 339.862,A -85,B 0,C 180,E1 -22115.383,E2 -22115.383} C_VEL
LIN {X 0,Y 185.675,Z 339.841,A -85,B 0,C 180,E1 -22121.134,E2 -22121.134} C_VEL
LIN {X 0,Y 185.725,Z 339.843,A -85,B 0,C 180,E1 -22124.64,E2 -22124.64} C_VEL
LIN {X 0,Y 185.943,Z 339.817,A -85,B 0,C 180,E1 -22129.329,E2 -22129.329} C_VEL
LIN {X 0,Y 185.967,Z 339.821,A -85,B 0,C 180,E1 -22133.491,E2 -22133.491} C_VEL
LIN {X 0,Y 186.21,Z 339.787,A -85,B 0,C 180,E1 -22137.838,E2 -22137.838} C_VEL
LIN {X 0,Y 186.409,Z 339.751,A -85,B 0,C 180,E1 -22140.001,E2 -22140.001} C_VEL
LIN {X 0,Y 185.928,Z 339.812,A -85,B 0,C 180,E1 -22144.336,E2 -22144.336} C_VEL
LIN {X 0,Y 185.975,Z 339.836,A -85,B 0,C 180,E1 -22147.465,E2 -22147.465} C_VEL
LIN {X 0,Y 186.723,Z 342.069,A -85,B 0,C 180,E1 -22148.251,E2 -22148.251} C_VEL
LIN {X 0,Y 188.462,Z 344.405,A -85,B 0,C 180,E1 -22149.67,E2 -22149.67} C_VEL
LIN {X 0,Y 190.505,Z 345.887,A -85,B 0,C 180,E1 -22151.101,E2 -22151.101} C_VEL
LIN {X 0,Y 192.152,Z 348.925,A -85,B 0,C 180,E1 -22152.342,E2 -22152.342} C_VEL
LIN {X 0,Y 194.703,Z 351.397,A -85,B 0,C 180,E1 -22153.932,E2 -22153.932} C_VEL
LIN {X 0,Y 196.942,Z 354.744,A -85,B 0,C 180,E1 -22155.293,E2 -22155.293} C_VEL
LIN {X 0,Y 198.513,Z 356.499,A -85,B 0,C 180,E1 -22156.156,E2 -22156.156} C_VEL
LIN {X 0,Y 201.309,Z 360.239,A -85,B 0,C 180,E1 -22157.639,E2 -22157.639} C_VEL
LIN {X 0,Y 205.425,Z 366.543,A -85,B 0,C 180,E1 -22159.681,E2 -22159.681} C_VEL
LIN {X 0,Y 209.959,Z 374.156,A -85,B 0,C 180,E1 -22161.757,E2 -22161.757} C_VEL
LIN {X 0,Y 216.228,Z 386.416,A -85,B 0,C 180,E1 -22164.406,E2 -22164.406} C_VEL
LIN {X 0,Y 220.811,Z 397.163,A -85,B 0,C 180,E1 -22166.228,E2 -22166.228} C_VEL
LIN {X 0,Y 217.572,Z 444.665,A -85,B 0,C 180,E1 -22167.768,E2 -22167.768} C_VEL
LIN {X 0,Y 216.473,Z 454.216,A -85,B 0,C 180,E1 -22168.234,E2 -22168.234} C_VEL
LIN {X 0,Y 214.834,Z 464.706,A -85,B 0,C 180,E1 -22168.975,E2 -22168.975} C_VEL
LIN {X 0,Y 212.684,Z 475.252,A -85,B 0,C 180,E1 -22169.979,E2 -22169.979} C_VEL
LIN {X 0,Y 210.371,Z 484.619,A -85,B 0,C 180,E1 -22171.122,E2 -22171.122} C_VEL
LIN {X 0,Y 207.588,Z 493.962,A -85,B 0,C 180,E1 -22172.535,E2 -22172.535} C_VEL
LIN {X 0,Y 204.349,Z 503.534,A -85,B 0,C 180,E1 -22174.37,E2 -22174.37} C_VEL
LIN {X 0,Y 200.973,Z 512.278,A -85,B 0,C 180,E1 -22176.457,E2 -22176.457} C_VEL
LIN {X 0,Y 197.849,Z 519.604,A -85,B 0,C 180,E1 -22178.604,E2 -22178.604} C_VEL
LIN {X 0,Y 195.027,Z 525.822,A -85,B 0,C 180,E1 -22180.821,E2 -22180.821} C_VEL
LIN {X 0,Y 191.865,Z 532.364,A -85,B 0,C 180,E1 -22183.765,E2 -22183.765} C_VEL
LIN {X 0,Y 189.306,Z 537.385,A -85,B 0,C 180,E1 -22186.622,E2 -22186.622} C_VEL
LIN {X 0,Y 186.78,Z 542.148,A -85,B 0,C 180,E1 -22190.234,E2 -22190.234} C_VEL
LIN {X 0,Y 185.426,Z 544.714,A -85,B 0,C 180,E1 -22192.745,E2 -22192.745} C_VEL
LIN {X 0,Y 184.418,Z 546.47,A -85,B 0,C 180,E1 -22195.136,E2 -22195.136} C_VEL
LIN {X 0,Y 183.65,Z 547.753,A -85,B 0,C 180,E1 -22197.605,E2 -22197.605} C_VEL
LIN {X 0,Y 183.052,Z 548.614,A -85,B 0,C 180,E1 -22200.059,E2 -22200.059} C_VEL
LIN {X 0,Y 182.731,Z 548.952,A -85,B 0,C 180,E1 -22202.514,E2 -22202.514} C_VEL
LIN {X 0,Y 182.538,Z 548.098,A -85,B 0,C 180,E1 -22207.356,E2 -22207.356} C_VEL
LIN {X 0,Y 182.717,Z 547.034,A -85,B 0,C 180,E1 -22209.747,E2 -22209.747} C_VEL
LIN {X 0,Y 183.354,Z 544.39,A -85,B 0,C 180,E1 -22213.388,E2 -22213.388} C_VEL
LIN {X 0,Y 184.21,Z 540.814,A -85,B 0,C 180,E1 -22216.767,E2 -22216.767} C_VEL
LIN {X 0,Y 185.732,Z 534.992,A -85,B 0,C 180,E1 -22220.722,E2 -22220.722} C_VEL
LIN {X 0,Y 187.234,Z 529.707,A -85,B 0,C 180,E1 -22223.535,E2 -22223.535} C_VEL
LIN {X 0,Y 189.071,Z 523.566,A -85,B 0,C 180,E1 -22226.188,E2 -22226.188} C_VEL
LIN {X 0,Y 191.398,Z 515.607,A -85,B 0,C 180,E1 -22228.948,E2 -22228.948} C_VEL
LIN {X 0,Y 193.654,Z 507.26,A -85,B 0,C 180,E1 -22231.3,E2 -22231.3} C_VEL
LIN {X 0,Y 196.054,Z 498.272,A -85,B 0,C 180,E1 -22233.34,E2 -22233.34} C_VEL
LIN {X 0,Y 198.055,Z 489.712,A -85,B 0,C 180,E1 -22234.943,E2 -22234.943} C_VEL
LIN {X 0,Y 200.224,Z 478.942,A -85,B 0,C 180,E1 -22236.551,E2 -22236.551} C_VEL
LIN {X 0,Y 202.021,Z 468.601,A -85,B 0,C 180,E1 -22237.748,E2 -22237.748} C_VEL
LIN {X 0,Y 203.363,Z 457.997,A -85,B 0,C 180,E1 -22238.696,E2 -22238.696} C_VEL
LIN {X 0,Y 204.496,Z 447.8,A -85,B 0,C 180,E1 -22239.333,E2 -22239.333} C_VEL
LIN {X 0,Y 205.609,Z 429.804,A -85,B 0,C 180,E1 -22240.031,E2 -22240.031} C_VEL
LIN {X 0,Y 207.644,Z 387.528,A -85,B 0,C 180,E1 -22241.471,E2 -22241.471} C_VEL
LIN {X 0,Y 199.536,Z 366.68,A -85,B 0,C 180,E1 -22243.774,E2 -22243.774} C_VEL
LIN {X 0,Y 193.099,Z 353.334,A -85,B 0,C 180,E1 -22245.625,E2 -22245.625} C_VEL
LIN {X 0,Y 187.503,Z 343.771,A -85,B 0,C 180,E1 -22247.258,E2 -22247.258} C_VEL
LIN {X 0,Y 185.899,Z 340.84,A -85,B 0,C 180,E1 -22247.836,E2 -22247.836} C_VEL
LIN {X 0,Y 185.698,Z 339.89,A -85,B 0,C 180,E1 -22248.413,E2 -22248.413} C_VEL
LIN {X 0,Y 185.581,Z 339.858,A -85,B 0,C 180,E1 -22252.254,E2 -22252.254} C_VEL
LIN {X 0,Y 185.561,Z 339.858,A -85,B 0,C 180,E1 -22257.033,E2 -22257.033} C_VEL
LIN {X 0,Y 185.58,Z 339.855,A -85,B 0,C 180,E1 -22259.493,E2 -22259.493} C_VEL
LIN {X 0,Y 185.52,Z 339.852,A -85,B 0,C 180,E1 -22264.628,E2 -22264.628} C_VEL
LIN {X 0,Y 185.546,Z 339.872,A -85,B 0,C 180,E1 -22267.304,E2 -22267.304} C_VEL
LIN {X 0,Y 185.487,Z 339.853,A -85,B 0,C 180,E1 -22270.73,E2 -22270.73} C_VEL
LIN {X 0,Y 185.483,Z 339.881,A -85,B 0,C 180,E1 -22276.048,E2 -22276.048} C_VEL
LIN {X 0,Y 185.469,Z 339.844,A -85,B 0,C 180,E1 -22279.895,E2 -22279.895} C_VEL
LIN {X 0,Y 185.508,Z 339.855,A -85,B 0,C 180,E1 -22282.711,E2 -22282.711} C_VEL
LIN {X 0,Y 185.533,Z 339.85,A -85,B 0,C 180,E1 -22287.972,E2 -22287.972} C_VEL
LIN {X 0,Y 185.549,Z 339.823,A -85,B 0,C 180,E1 -22290.595,E2 -22290.595} C_VEL
LIN {X 0,Y 185.582,Z 339.866,A -85,B 0,C 180,E1 -22295.381,E2 -22295.381} C_VEL
LIN {X 0,Y 185.636,Z 339.809,A -85,B 0,C 180,E1 -22301.17,E2 -22301.17} C_VEL
LIN {X 0,Y 185.674,Z 339.828,A -85,B 0,C 180,E1 -22304.635,E2 -22304.635} C_VEL
LIN {X 0,Y 185.89,Z 339.82,A -85,B 0,C 180,E1 -22309.419,E2 -22309.419} C_VEL
LIN {X 0,Y 185.932,Z 339.771,A -85,B 0,C 180,E1 -22313.488,E2 -22313.488} C_VEL
LIN {X 0,Y 186.179,Z 339.784,A -85,B 0,C 180,E1 -22317.836,E2 -22317.836} C_VEL
LIN {X 0,Y 186.383,Z 339.766,A -85,B 0,C 180,E1 -22319.999,E2 -22319.999} C_VEL
LIN {X 0,Y 185.888,Z 339.783,A -85,B 0,C 180,E1 -22324.336,E2 -22324.336} C_VEL
LIN {X 0,Y 185.981,Z 339.812,A -85,B 0,C 180,E1 -22328.693,E2 -22328.693} C_VEL
LIN {X 0,Y 185.701,Z 339.827,A -85,B 0,C 180,E1 -22333.124,E2 -22333.124} C_VEL
LIN {X 0,Y 185.626,Z 339.861,A -85,B 0,C 180,E1 -22338.821,E2 -22338.821} C_VEL
LIN {X 0,Y 185.578,Z 339.839,A -85,B 0,C 180,E1 -22344.645,E2 -22344.645} C_VEL
LIN {X 0,Y 185.544,Z 339.86,A -85,B 0,C 180,E1 -22349.498,E2 -22349.498} C_VEL
LIN {X 0,Y 185.496,Z 339.88,A -85,B 0,C 180,E1 -22354.632,E2 -22354.632} C_VEL
LIN {X 0,Y 185.499,Z 339.861,A -85,B 0,C 180,E1 -22357.314,E2 -22357.314} C_VEL
LIN {X 0,Y 185.459,Z 339.88,A -85,B 0,C 180,E1 -22360.72,E2 -22360.72} C_VEL
LIN {X 0,Y 185.454,Z 339.877,A -85,B 0,C 180,E1 -22366.056,E2 -22366.056} C_VEL
LIN {X 0,Y 185.482,Z 340.122,A -85,B 0,C 180,E1 -22366.797,E2 -22366.797} C_VEL
LIN {X 0,Y 186.105,Z 342.392,A -85,B 0,C 180,E1 -22368.113,E2 -22368.113} C_VEL
LIN {X 0,Y 190.05,Z 350.126,A -85,B 0,C 180,E1 -22369.419,E2 -22369.419} C_VEL
LIN {X 0,Y 196.029,Z 362.451,A -85,B 0,C 180,E1 -22371.203,E2 -22371.203} C_VEL
LIN {X 0,Y 203.724,Z 381.255,A -85,B 0,C 180,E1 -22373.431,E2 -22373.431} C_VEL
LIN {X 0,Y 206.35,Z 389.051,A -85,B 0,C 180,E1 -22374.208,E2 -22374.208} C_VEL
LIN {X 0,Y 207.302,Z 397.014,A -85,B 0,C 180,E1 -22374.699,E2 -22374.699} C_VEL
LIN {X 0,Y 205.671,Z 429.883,A -85,B 0,C 180,E1 -22375.811,E2 -22375.811} C_VEL
LIN {X 0,Y 204.738,Z 435.721,A -85,B 0,C 180,E1 -22375.901,E2 -22375.901} C_VEL
LIN {X 0,Y 198.469,Z 454.545,A -85,B 0,C 180,E1 -22375.868,E2 -22375.868} C_VEL
LIN {X 0,Y 197.62,Z 458.349,A -85,B 0,C 180,E1 -22376.048,E2 -22376.048} C_VEL
LIN {X 0,Y 197.405,Z 460.252,A -85,B 0,C 180,E1 -22376.188,E2 -22376.188} C_VEL
LIN {X 0,Y 195.961,Z 470.311,A -85,B 0,C 180,E1 -22376.996,E2 -22376.996} C_VEL
LIN {X 0,Y 194.253,Z 480.159,A -85,B 0,C 180,E1 -22378.053,E2 -22378.053} C_VEL
LIN {X 0,Y 192.557,Z 489.047,A -85,B 0,C 180,E1 -22379.271,E2 -22379.271} C_VEL
LIN {X 0,Y 190.094,Z 499.081,A -85,B 0,C 180,E1 -22380.971,E2 -22380.971} C_VEL
LIN {X 0,Y 187.625,Z 508.494,A -85,B 0,C 180,E1 -22382.988,E2 -22382.988} C_VEL
LIN {X 0,Y 185.716,Z 515.531,A -85,B 0,C 180,E1 -22384.803,E2 -22384.803} C_VEL
LIN {X 0,Y 183.36,Z 523.877,A -85,B 0,C 180,E1 -22387.462,E2 -22387.462} C_VEL
LIN {X 0,Y 181.204,Z 530.803,A -85,B 0,C 180,E1 -22390.161,E2 -22390.161} C_VEL
LIN {X 0,Y 179.419,Z 536.585,A -85,B 0,C 180,E1 -22392.915,E2 -22392.915} C_VEL
LIN {X 0,Y 177.819,Z 542.175,A -85,B 0,C 180,E1 -22396.282,E2 -22396.282} C_VEL
LIN {X 0,Y 176.783,Z 546.56,A -85,B 0,C 180,E1 -22399.694,E2 -22399.694} C_VEL
LIN {X 0,Y 176.15,Z 549.854,A -85,B 0,C 180,E1 -22403.125,E2 -22403.125} C_VEL
LIN {X 0,Y 175.939,Z 551.482,A -85,B 0,C 180,E1 -22405.417,E2 -22405.417} C_VEL
LIN {X 0,Y 175.972,Z 553.507,A -85,B 0,C 180,E1 -22410,E2 -22410} C_VEL
LIN {X 0,Y 175.908,Z 553.882,A -85,B 0,C 180,E1 -22412.805,E2 -22412.805} C_VEL
LIN {X 0,Y 176.232,Z 553.45,A -85,B 0,C 180,E1 -22416.871,E2 -22416.871} C_VEL
LIN {X 0,Y 177.2,Z 551.388,A -85,B 0,C 180,E1 -22421.438,E2 -22421.438} C_VEL
LIN {X 0,Y 178.575,Z 548.813,A -85,B 0,C 180,E1 -22424.822,E2 -22424.822} C_VEL
LIN {X 0,Y 180.458,Z 545.241,A -85,B 0,C 180,E1 -22428.153,E2 -22428.153} C_VEL
LIN {X 0,Y 183.126,Z 540.568,A -85,B 0,C 180,E1 -22431.382,E2 -22431.382} C_VEL
LIN {X 0,Y 186.092,Z 534.672,A -85,B 0,C 180,E1 -22434.546,E2 -22434.546} C_VEL
LIN {X 0,Y 189.642,Z 527.341,A -85,B 0,C 180,E1 -22437.596,E2 -22437.596} C_VEL
LIN {X 0,Y 193.109,Z 519.93,A -85,B 0,C 180,E1 -22440.027,E2 -22440.027} C_VEL
LIN {X 0,Y 196.555,Z 511.956,A -85,B 0,C 180,E1 -22442.132,E2 -22442.132} C_VEL
LIN {X 0,Y 199.798,Z 503.524,A -85,B 0,C 180,E1 -22443.946,E2 -22443.946} C_VEL
LIN {X 0,Y 203.274,Z 493.252,A -85,B 0,C 180,E1 -22445.692,E2 -22445.692} C_VEL
LIN {X 0,Y 205.984,Z 483.866,A -85,B 0,C 180,E1 -22446.967,E2 -22446.967} C_VEL
LIN {X 0,Y 208.555,Z 473.061,A -85,B 0,C 180,E1 -22448.105,E2 -22448.105} C_VEL
LIN {X 0,Y 210.539,Z 462.889,A -85,B 0,C 180,E1 -22448.901,E2 -22448.901} C_VEL
LIN {X 0,Y 212.134,Z 451.651,A -85,B 0,C 180,E1 -22449.524,E2 -22449.524} C_VEL
LIN {X 0,Y 213.557,Z 432.499,A -85,B 0,C 180,E1 -22450.233,E2 -22450.233} C_VEL
LIN {X 0,Y 215.486,Z 403.2,A -85,B 0,C 180,E1 -22451.185,E2 -22451.185} C_VEL
LIN {X 0,Y 211.207,Z 392.22,A -85,B 0,C 180,E1 -22453.07,E2 -22453.07} C_VEL
LIN {X 0,Y 206.204,Z 381.753,A -85,B 0,C 180,E1 -22455.349,E2 -22455.349} C_VEL
LIN {X 0,Y 201.119,Z 372.672,A -85,B 0,C 180,E1 -22457.868,E2 -22457.868} C_VEL
LIN {X 0,Y 197.653,Z 366.97,A -85,B 0,C 180,E1 -22459.739,E2 -22459.739} C_VEL
LIN {X 0,Y 195.168,Z 363.071,A -85,B 0,C 180,E1 -22461.195,E2 -22461.195} C_VEL
LIN {X 0,Y 191.802,Z 358.115,A -85,B 0,C 180,E1 -22463.32,E2 -22463.32} C_VEL
LIN {X 0,Y 187.705,Z 352.46,A -85,B 0,C 180,E1 -22466.295,E2 -22466.295} C_VEL
LIN {X 0,Y 184.492,Z 348.978,A -85,B 0,C 180,E1 -22468.893,E2 -22468.893} C_VEL
LIN {X 0,Y 183.287,Z 346.611,A -85,B 0,C 180,E1 -22470.102,E2 -22470.102} C_VEL
LIN {X 0,Y 180.495,Z 344.812,A -85,B 0,C 180,E1 -22472.931,E2 -22472.931} C_VEL
LIN {X 0,Y 179.017,Z 342.584,A -85,B 0,C 180,E1 -22474.896,E2 -22474.896} C_VEL
LIN {X 0,Y 178.533,Z 340.735,A -85,B 0,C 180,E1 -22475.968,E2 -22475.968} C_VEL
LIN {X 0,Y 178.65,Z 340.715,A -85,B 0,C 180,E1 -22481.657,E2 -22481.657} C_VEL
LIN {X 0,Y 178.688,Z 340.71,A -85,B 0,C 180,E1 -22486.351,E2 -22486.351} C_VEL
LIN {X 0,Y 178.976,Z 340.674,A -85,B 0,C 180,E1 -22490.964,E2 -22490.964} C_VEL
LIN {X 0,Y 179.156,Z 340.664,A -85,B 0,C 180,E1 -22497.752,E2 -22497.752} C_VEL
LIN {X 0,Y 179.372,Z 340.627,A -85,B 0,C 180,E1 -22500.001,E2 -22500.001} C_VEL
LIN {X 0,Y 179.244,Z 340.819,A -85,B 0,C 180,E1 -22501.335,E2 -22501.335} C_VEL
LIN {X 0,Y 180.004,Z 343.354,A -85,B 0,C 180,E1 -22502.588,E2 -22502.588} C_VEL
LIN {X 0,Y 181.547,Z 345.402,A -85,B 0,C 180,E1 -22504.441,E2 -22504.441} C_VEL
LIN {X 0,Y 184.008,Z 346.889,A -85,B 0,C 180,E1 -22506.764,E2 -22506.764} C_VEL
LIN {X 0,Y 185.846,Z 350.195,A -85,B 0,C 180,E1 -22508.475,E2 -22508.475} C_VEL
LIN {X 0,Y 188.324,Z 352.437,A -85,B 0,C 180,E1 -22510.354,E2 -22510.354} C_VEL
LIN {X 0,Y 190.39,Z 355.742,A -85,B 0,C 180,E1 -22511.917,E2 -22511.917} C_VEL
LIN {X 0,Y 192.274,Z 357.649,A -85,B 0,C 180,E1 -22513.151,E2 -22513.151} C_VEL
LIN {X 0,Y 194.865,Z 361.332,A -85,B 0,C 180,E1 -22514.773,E2 -22514.773} C_VEL
LIN {X 0,Y 196.149,Z 363,A -85,B 0,C 180,E1 -22515.521,E2 -22515.521} C_VEL
LIN {X 0,Y 199.924,Z 368.353,A -85,B 0,C 180,E1 -22517.602,E2 -22517.602} C_VEL
LIN {X 0,Y 204.167,Z 375.195,A -85,B 0,C 180,E1 -22519.742,E2 -22519.742} C_VEL
LIN {X 0,Y 209.734,Z 385.777,A -85,B 0,C 180,E1 -22522.341,E2 -22522.341} C_VEL
LIN {X 0,Y 214.342,Z 395.896,A -85,B 0,C 180,E1 -22524.342,E2 -22524.342} C_VEL
LIN {X 0,Y 215.716,Z 399.478,A -85,B 0,C 180,E1 -22524.937,E2 -22524.937} C_VEL
LIN {X 0,Y 212.55,Z 444.656,A -85,B 0,C 180,E1 -22526.435,E2 -22526.435} C_VEL
LIN {X 0,Y 211.405,Z 454.299,A -85,B 0,C 180,E1 -22526.909,E2 -22526.909} C_VEL
LIN {X 0,Y 209.863,Z 463.861,A -85,B 0,C 180,E1 -22527.57,E2 -22527.57} C_VEL
LIN {X 0,Y 207.623,Z 474.714,A -85,B 0,C 180,E1 -22528.6,E2 -22528.6} C_VEL
LIN {X 0,Y 205.304,Z 483.842,A -85,B 0,C 180,E1 -22529.699,E2 -22529.699} C_VEL
LIN {X 0,Y 202.472,Z 493.073,A -85,B 0,C 180,E1 -22531.075,E2 -22531.075} C_VEL
LIN {X 0,Y 198.982,Z 503.028,A -85,B 0,C 180,E1 -22532.982,E2 -22532.982} C_VEL
LIN {X 0,Y 195.337,Z 512.041,A -85,B 0,C 180,E1 -22535.146,E2 -22535.146} C_VEL
LIN {X 0,Y 192.105,Z 519.256,A -85,B 0,C 180,E1 -22537.278,E2 -22537.278} C_VEL
LIN {X 0,Y 189.047,Z 525.607,A -85,B 0,C 180,E1 -22539.568,E2 -22539.568} C_VEL
LIN {X 0,Y 185.996,Z 531.643,A -85,B 0,C 180,E1 -22542.283,E2 -22542.283} C_VEL
LIN {X 0,Y 183.493,Z 536.297,A -85,B 0,C 180,E1 -22544.881,E2 -22544.881} C_VEL
LIN {X 0,Y 180.636,Z 541.402,A -85,B 0,C 180,E1 -22548.592,E2 -22548.592} C_VEL
LIN {X 0,Y 178.699,Z 544.708,A -85,B 0,C 180,E1 -22551.867,E2 -22551.867} C_VEL
LIN {X 0,Y 176.844,Z 547.656,A -85,B 0,C 180,E1 -22556.572,E2 -22556.572} C_VEL
LIN {X 0,Y 176.212,Z 548.556,A -85,B 0,C 180,E1 -22558.769,E2 -22558.769} C_VEL
LIN {X 0,Y 175.713,Z 548.985,A -85,B 0,C 180,E1 -22561.635,E2 -22561.635} C_VEL
LIN {X 0,Y 175.412,Z 548.53,A -85,B 0,C 180,E1 -22566.381,E2 -22566.381} C_VEL
LIN {X 0,Y 175.528,Z 547.483,A -85,B 0,C 180,E1 -22568.878,E2 -22568.878} C_VEL
LIN {X 0,Y 176.349,Z 544.202,A -85,B 0,C 180,E1 -22573.801,E2 -22573.801} C_VEL
LIN {X 0,Y 177.301,Z 540.391,A -85,B 0,C 180,E1 -22577.408,E2 -22577.408} C_VEL
LIN {X 0,Y 178.691,Z 535.358,A -85,B 0,C 180,E1 -22580.949,E2 -22580.949} C_VEL
LIN {X 0,Y 180.223,Z 530.187,A -85,B 0,C 180,E1 -22583.844,E2 -22583.844} C_VEL
LIN {X 0,Y 182.257,Z 523.6,A -85,B 0,C 180,E1 -22586.795,E2 -22586.795} C_VEL
LIN {X 0,Y 184.523,Z 516.252,A -85,B 0,C 180,E1 -22589.455,E2 -22589.455} C_VEL
LIN {X 0,Y 187.11,Z 506.957,A -85,B 0,C 180,E1 -22592.153,E2 -22592.153} C_VEL
LIN {X 0,Y 189.308,Z 499.163,A -85,B 0,C 180,E1 -22593.992,E2 -22593.992} C_VEL
LIN {X 0,Y 191.79,Z 488.956,A -85,B 0,C 180,E1 -22595.939,E2 -22595.939} C_VEL
LIN {X 0,Y 193.644,Z 480.214,A -85,B 0,C 180,E1 -22597.298,E2 -22597.298} C_VEL
LIN {X 0,Y 195.668,Z 468.985,A -85,B 0,C 180,E1 -22598.651,E2 -22598.651} C_VEL
LIN {X 0,Y 197.057,Z 458.491,A -85,B 0,C 180,E1 -22599.624,E2 -22599.624} C_VEL
LIN {X 0,Y 198.342,Z 446.849,A -85,B 0,C 180,E1 -22600.354,E2 -22600.354} C_VEL
LIN {X 0,Y 199.534,Z 428.315,A -85,B 0,C 180,E1 -22601.071,E2 -22601.071} C_VEL
LIN {X 0,Y 201.426,Z 388.824,A -85,B 0,C 180,E1 -22602.464,E2 -22602.464} C_VEL
LIN {X 0,Y 193.585,Z 368.921,A -85,B 0,C 180,E1 -22604.799,E2 -22604.799} C_VEL
LIN {X 0,Y 187.591,Z 356.648,A -85,B 0,C 180,E1 -22606.61,E2 -22606.61} C_VEL
LIN {X 0,Y 182.732,Z 348.379,A -85,B 0,C 180,E1 -22608.094,E2 -22608.094} C_VEL
LIN {X 0,Y 180.354,Z 344.546,A -85,B 0,C 180,E1 -22608.849,E2 -22608.849} C_VEL
LIN {X 0,Y 178.837,Z 341.921,A -85,B 0,C 180,E1 -22609.409,E2 -22609.409} C_VEL
LIN {X 0,Y 178.579,Z 340.803,A -85,B 0,C 180,E1 -22610.003,E2 -22610.003} C_VEL
LIN {X 0,Y 178.504,Z 340.751,A -85,B 0,C 180,E1 -22615.664,E2 -22615.664} C_VEL
LIN {X 0,Y 178.501,Z 340.75,A -85,B 0,C 180,E1 -22620.787,E2 -22620.787} C_VEL
LIN {X 0,Y 178.497,Z 340.726,A -85,B 0,C 180,E1 -22624.224,E2 -22624.224} C_VEL
LIN {X 0,Y 178.42,Z 340.752,A -85,B 0,C 180,E1 -22629.068,E2 -22629.068} C_VEL
LIN {X 0,Y 178.406,Z 340.731,A -85,B 0,C 180,E1 -22632.043,E2 -22632.043} C_VEL
LIN {X 0,Y 178.41,Z 340.761,A -85,B 0,C 180,E1 -22635.159,E2 -22635.159} C_VEL
LIN {X 0,Y 178.41,Z 340.735,A -85,B 0,C 180,E1 -22638.457,E2 -22638.457} C_VEL
LIN {X 0,Y 178.424,Z 340.75,A -85,B 0,C 180,E1 -22643.783,E2 -22643.783} C_VEL
LIN {X 0,Y 178.486,Z 340.746,A -85,B 0,C 180,E1 -22646.546,E2 -22646.546} C_VEL
LIN {X 0,Y 178.445,Z 340.712,A -85,B 0,C 180,E1 -22651.795,E2 -22651.795} C_VEL
LIN {X 0,Y 178.517,Z 340.743,A -85,B 0,C 180,E1 -22654.889,E2 -22654.889} C_VEL
LIN {X 0,Y 178.566,Z 340.69,A -85,B 0,C 180,E1 -22660.839,E2 -22660.839} C_VEL
LIN {X 0,Y 178.649,Z 340.726,A -85,B 0,C 180,E1 -22666.347,E2 -22666.347} C_VEL
LIN {X 0,Y 178.906,Z 340.669,A -85,B 0,C 180,E1 -22670.959,E2 -22670.959} C_VEL
LIN {X 0,Y 179.126,Z 340.663,A -85,B 0,C 180,E1 -22677.751,E2 -22677.751} C_VEL
LIN {X 0,Y 179.348,Z 340.642,A -85,B 0,C 180,E1 -22679.999,E2 -22679.999} C_VEL
LIN {X 0,Y 178.838,Z 340.66,A -85,B 0,C 180,E1 -22684.507,E2 -22684.507} C_VEL
LIN {X 0,Y 178.91,Z 340.694,A -85,B 0,C 180,E1 -22689.04,E2 -22689.04} C_VEL
LIN {X 0,Y 178.627,Z 340.701,A -85,B 0,C 180,E1 -22693.654,E2 -22693.654} C_VEL
LIN {X 0,Y 178.555,Z 340.743,A -85,B 0,C 180,E1 -22699.151,E2 -22699.151} C_VEL
LIN {X 0,Y 178.516,Z 340.721,A -85,B 0,C 180,E1 -22705.11,E2 -22705.11} C_VEL
LIN {X 0,Y 178.46,Z 340.732,A -85,B 0,C 180,E1 -22710.794,E2 -22710.794} C_VEL
LIN {X 0,Y 178.482,Z 340.754,A -85,B 0,C 180,E1 -22714.217,E2 -22714.217} C_VEL
LIN {X 0,Y 178.386,Z 340.756,A -85,B 0,C 180,E1 -22719.076,E2 -22719.076} C_VEL
LIN {X 0,Y 178.391,Z 340.75,A -85,B 0,C 180,E1 -22722.046,E2 -22722.046} C_VEL
LIN {X 0,Y 178.413,Z 340.931,A -85,B 0,C 180,E1 -22725.558,E2 -22725.558} C_VEL
LIN {X 0,Y 178.83,Z 342.476,A -85,B 0,C 180,E1 -22726.434,E2 -22726.434} C_VEL
LIN {X 0,Y 185.883,Z 355.951,A -85,B 0,C 180,E1 -22728.818,E2 -22728.818} C_VEL
LIN {X 0,Y 191.886,Z 368.864,A -85,B 0,C 180,E1 -22730.688,E2 -22730.688} C_VEL
LIN {X 0,Y 198.264,Z 384.886,A -85,B 0,C 180,E1 -22732.633,E2 -22732.633} C_VEL
LIN {X 0,Y 200.413,Z 391.399,A -85,B 0,C 180,E1 -22733.3,E2 -22733.3} C_VEL
LIN {X 0,Y 201.166,Z 397.745,A -85,B 0,C 180,E1 -22733.706,E2 -22733.706} C_VEL
LIN {X 0,Y 198.394,Z 449.296,A -85,B 0,C 180,E1 -22735.55,E2 -22735.55} C_VEL
LIN {X 0,Y 197.592,Z 458.747,A -85,B 0,C 180,E1 -22736.084,E2 -22736.084} C_VEL
LIN {X 0,Y 197.405,Z 460.252,A -85,B 0,C 180,E1 -22736.188,E2 -22736.188} C_VEL
LIN {X 0,Y 196.354,Z 464.05,A -85,B 0,C 180,E1 -22736.357,E2 -22736.357} C_VEL
LIN {X 0,Y 192.962,Z 469.901,A -85,B 0,C 180,E1 -22736.458,E2 -22736.458} C_VEL
LIN {X 0,Y 189.371,Z 475.625,A -85,B 0,C 180,E1 -22736.627,E2 -22736.627} C_VEL
LIN {X 0,Y 188.387,Z 478.015,A -85,B 0,C 180,E1 -22736.828,E2 -22736.828} C_VEL
LIN {X 0,Y 188.098,Z 479.223,A -85,B 0,C 180,E1 -22736.979,E2 -22736.979} C_VEL
LIN {X 0,Y 186.079,Z 489.299,A -85,B 0,C 180,E1 -22738.396,E2 -22738.396} C_VEL
LIN {X 0,Y 183.527,Z 499.27,A -85,B 0,C 180,E1 -22740.144,E2 -22740.144} C_VEL
LIN {X 0,Y 181.276,Z 507.605,A -85,B 0,C 180,E1 -22741.96,E2 -22741.96} C_VEL
LIN {X 0,Y 178.747,Z 516.499,A -85,B 0,C 180,E1 -22744.373,E2 -22744.373} C_VEL
LIN {X 0,Y 176.709,Z 523.223,A -85,B 0,C 180,E1 -22746.564,E2 -22746.564} C_VEL
LIN {X 0,Y 174.472,Z 530.248,A -85,B 0,C 180,E1 -22749.362,E2 -22749.362} C_VEL
LIN {X 0,Y 172.627,Z 536.113,A -85,B 0,C 180,E1 -22752.221,E2 -22752.221} C_VEL
LIN {X 0,Y 170.897,Z 541.784,A -85,B 0,C 180,E1 -22755.715,E2 -22755.715} C_VEL
LIN {X 0,Y 169.768,Z 546.24,A -85,B 0,C 180,E1 -22759.263,E2 -22759.263} C_VEL
LIN {X 0,Y 169.107,Z 549.6,A -85,B 0,C 180,E1 -22762.838,E2 -22762.838} C_VEL
LIN {X 0,Y 168.858,Z 551.228,A -85,B 0,C 180,E1 -22765.225,E2 -22765.225} C_VEL
LIN {X 0,Y 168.87,Z 553.362,A -85,B 0,C 180,E1 -22770,E2 -22770} C_VEL
LIN {X 0,Y 168.87,Z 553.721,A -85,B 0,C 180,E1 -22774.774,E2 -22774.774} C_VEL
LIN {X 0,Y 169.165,Z 553.382,A -85,B 0,C 180,E1 -22777.159,E2 -22777.159} C_VEL
LIN {X 0,Y 170.243,Z 551.44,A -85,B 0,C 180,E1 -22781.912,E2 -22781.912} C_VEL
LIN {X 0,Y 171.707,Z 548.924,A -85,B 0,C 180,E1 -22785.429,E2 -22785.429} C_VEL
LIN {X 0,Y 173.729,Z 545.421,A -85,B 0,C 180,E1 -22788.882,E2 -22788.882} C_VEL
LIN {X 0,Y 176.539,Z 540.838,A -85,B 0,C 180,E1 -22792.222,E2 -22792.222} C_VEL
LIN {X 0,Y 180.427,Z 533.545,A -85,B 0,C 180,E1 -22796.173,E2 -22796.173} C_VEL
LIN {X 0,Y 183.41,Z 527.823,A -85,B 0,C 180,E1 -22798.619,E2 -22798.619} C_VEL
LIN {X 0,Y 187.03,Z 520.525,A -85,B 0,C 180,E1 -22801.11,E2 -22801.11} C_VEL
LIN {X 0,Y 191.035,Z 511.677,A -85,B 0,C 180,E1 -22803.493,E2 -22803.493} C_VEL
LIN {X 0,Y 193.999,Z 504.422,A -85,B 0,C 180,E1 -22805.107,E2 -22805.107} C_VEL
LIN {X 0,Y 197.607,Z 494.365,A -85,B 0,C 180,E1 -22806.882,E2 -22806.882} C_VEL
LIN {X 0,Y 200.909,Z 483.469,A -85,B 0,C 180,E1 -22808.383,E2 -22808.383} C_VEL
LIN {X 0,Y 203.336,Z 473.794,A -85,B 0,C 180,E1 -22809.428,E2 -22809.428} C_VEL
LIN {X 0,Y 205.656,Z 462.354,A -85,B 0,C 180,E1 -22810.328,E2 -22810.328} C_VEL
LIN {X 0,Y 207.236,Z 451.659,A -85,B 0,C 180,E1 -22810.924,E2 -22810.924} C_VEL
LIN {X 0,Y 208.637,Z 433.768,A -85,B 0,C 180,E1 -22811.607,E2 -22811.607} C_VEL
LIN {X 0,Y 210.606,Z 405.425,A -85,B 0,C 180,E1 -22812.536,E2 -22812.536} C_VEL
LIN {X 0,Y 206.516,Z 395.16,A -85,B 0,C 180,E1 -22814.449,E2 -22814.449} C_VEL
LIN {X 0,Y 202.46,Z 386.35,A -85,B 0,C 180,E1 -22816.46,E2 -22816.46} C_VEL
LIN {X 0,Y 197.795,Z 377.832,A -85,B 0,C 180,E1 -22818.91,E2 -22818.91} C_VEL
LIN {X 0,Y 194.496,Z 372.164,A -85,B 0,C 180,E1 -22820.84,E2 -22820.84} C_VEL
LIN {X 0,Y 192.484,Z 368.942,A -85,B 0,C 180,E1 -22822.09,E2 -22822.09} C_VEL
LIN {X 0,Y 189.28,Z 364.015,A -85,B 0,C 180,E1 -22824.254,E2 -22824.254} C_VEL
LIN {X 0,Y 185.531,Z 358.657,A -85,B 0,C 180,E1 -22827.132,E2 -22827.132} C_VEL
LIN {X 0,Y 182.662,Z 355.485,A -85,B 0,C 180,E1 -22829.59,E2 -22829.59} C_VEL
LIN {X 0,Y 181.556,Z 353.354,A -85,B 0,C 180,E1 -22830.768,E2 -22830.768} C_VEL
LIN {X 0,Y 178.796,Z 351.316,A -85,B 0,C 180,E1 -22833.756,E2 -22833.756} C_VEL
LIN {X 0,Y 177.331,Z 348.731,A -85,B 0,C 180,E1 -22835.906,E2 -22835.906} C_VEL
LIN {X 0,Y 176.951,Z 347.66,A -85,B 0,C 180,E1 -22836.599,E2 -22836.599} C_VEL
LIN {X 0,Y 173.222,Z 345.187,A -85,B 0,C 180,E1 -22846.838,E2 -22846.838} C_VEL
LIN {X 0,Y 173.401,Z 345.101,A -85,B 0,C 180,E1 -22850.671,E2 -22850.671} C_VEL
LIN {X 0,Y 177.651,Z 347.671,A -85,B 0,C 180,E1 -22860.567,E2 -22860.567} C_VEL
LIN {X 0,Y 178.801,Z 350.613,A -85,B 0,C 180,E1 -22862.394,E2 -22862.394} C_VEL
LIN {X 0,Y 180.816,Z 352.728,A -85,B 0,C 180,E1 -22864.738,E2 -22864.738} C_VEL
LIN {X 0,Y 182.231,Z 353.642,A -85,B 0,C 180,E1 -22866.089,E2 -22866.089} C_VEL
LIN {X 0,Y 184.129,Z 356.883,A -85,B 0,C 180,E1 -22867.949,E2 -22867.949} C_VEL
LIN {X 0,Y 186.261,Z 358.996,A -85,B 0,C 180,E1 -22869.647,E2 -22869.647} C_VEL
LIN {X 0,Y 188.587,Z 362.468,A -85,B 0,C 180,E1 -22871.445,E2 -22871.445} C_VEL
LIN {X 0,Y 189.997,Z 364.057,A -85,B 0,C 180,E1 -22872.416,E2 -22872.416} C_VEL
LIN {X 0,Y 194.012,Z 369.741,A -85,B 0,C 180,E1 -22874.99,E2 -22874.99} C_VEL
LIN {X 0,Y 197.588,Z 374.902,A -85,B 0,C 180,E1 -22877.043,E2 -22877.043} C_VEL
LIN {X 0,Y 202.751,Z 384.013,A -85,B 0,C 180,E1 -22879.753,E2 -22879.753} C_VEL
LIN {X 0,Y 208.122,Z 395.243,A -85,B 0,C 180,E1 -22882.344,E2 -22882.344} C_VEL
LIN {X 0,Y 210.82,Z 401.846,A -85,B 0,C 180,E1 -22883.581,E2 -22883.581} C_VEL
LIN {X 0,Y 207.711,Z 444.491,A -85,B 0,C 180,E1 -22885.021,E2 -22885.021} C_VEL
LIN {X 0,Y 206.489,Z 454.441,A -85,B 0,C 180,E1 -22885.514,E2 -22885.514} C_VEL
LIN {X 0,Y 204.705,Z 464.75,A -85,B 0,C 180,E1 -22886.243,E2 -22886.243} C_VEL
LIN {X 0,Y 202.507,Z 474.83,A -85,B 0,C 180,E1 -22887.213,E2 -22887.213} C_VEL
LIN {X 0,Y 199.831,Z 484.778,A -85,B 0,C 180,E1 -22888.449,E2 -22888.449} C_VEL
LIN {X 0,Y 196.48,Z 494.961,A -85,B 0,C 180,E1 -22890.052,E2 -22890.052} C_VEL
LIN {X 0,Y 193.241,Z 503.664,A -85,B 0,C 180,E1 -22891.774,E2 -22891.774} C_VEL
LIN {X 0,Y 189.879,Z 511.679,A -85,B 0,C 180,E1 -22893.725,E2 -22893.725} C_VEL
LIN {X 0,Y 186.479,Z 518.93,A -85,B 0,C 180,E1 -22895.876,E2 -22895.876} C_VEL
LIN {X 0,Y 182.823,Z 526.043,A -85,B 0,C 180,E1 -22898.513,E2 -22898.513} C_VEL
LIN {X 0,Y 179.106,Z 532.876,A -85,B 0,C 180,E1 -22901.794,E2 -22901.794} C_VEL
LIN {X 0,Y 176.697,Z 537.085,A -85,B 0,C 180,E1 -22904.28,E2 -22904.28} C_VEL
LIN {X 0,Y 173.726,Z 541.964,A -85,B 0,C 180,E1 -22908.126,E2 -22908.126} C_VEL
LIN {X 0,Y 172.009,Z 544.701,A -85,B 0,C 180,E1 -22910.925,E2 -22910.925} C_VEL
LIN {X 0,Y 170.306,Z 547.252,A -85,B 0,C 180,E1 -22914.709,E2 -22914.709} C_VEL
LIN {X 0,Y 169.478,Z 548.324,A -85,B 0,C 180,E1 -22917.379,E2 -22917.379} C_VEL
LIN {X 0,Y 168.474,Z 549.156,A -85,B 0,C 180,E1 -22922.686,E2 -22922.686} C_VEL
LIN {X 0,Y 168.323,Z 548.425,A -85,B 0,C 180,E1 -22926.719,E2 -22926.719} C_VEL
LIN {X 0,Y 168.584,Z 546.705,A -85,B 0,C 180,E1 -22930.518,E2 -22930.518} C_VEL
LIN {X 0,Y 169.344,Z 543.867,A -85,B 0,C 180,E1 -22934.35,E2 -22934.35} C_VEL
LIN {X 0,Y 170.379,Z 539.918,A -85,B 0,C 180,E1 -22938.098,E2 -22938.098} C_VEL
LIN {X 0,Y 171.32,Z 536.695,A -85,B 0,C 180,E1 -22940.556,E2 -22940.556} C_VEL
LIN {X 0,Y 173.201,Z 530.633,A -85,B 0,C 180,E1 -22944.178,E2 -22944.178} C_VEL
LIN {X 0,Y 175.681,Z 522.926,A -85,B 0,C 180,E1 -22947.708,E2 -22947.708} C_VEL
LIN {X 0,Y 178.147,Z 515.084,A -85,B 0,C 180,E1 -22950.565,E2 -22950.565} C_VEL
LIN {X 0,Y 180.337,Z 507.653,A -85,B 0,C 180,E1 -22952.792,E2 -22952.792} C_VEL
LIN {X 0,Y 182.716,Z 499.508,A -85,B 0,C 180,E1 -22954.792,E2 -22954.792} C_VEL
LIN {X 0,Y 185.296,Z 489.296,A -85,B 0,C 180,E1 -22956.807,E2 -22956.807} C_VEL
LIN {X 0,Y 187.432,Z 479.484,A -85,B 0,C 180,E1 -22958.355,E2 -22958.355} C_VEL
LIN {X 0,Y 189.374,Z 469.233,A -85,B 0,C 180,E1 -22959.614,E2 -22959.614} C_VEL
LIN {X 0,Y 190.901,Z 458.055,A -85,B 0,C 180,E1 -22960.667,E2 -22960.667} C_VEL
LIN {X 0,Y 192.158,Z 447.099,A -85,B 0,C 180,E1 -22961.368,E2 -22961.368} C_VEL
LIN {X 0,Y 193.429,Z 428.085,A -85,B 0,C 180,E1 -22962.119,E2 -22962.119} C_VEL
LIN {X 0,Y 195.32,Z 390.82,A -85,B 0,C 180,E1 -22963.463,E2 -22963.463} C_VEL
LIN {X 0,Y 188.18,Z 372.362,A -85,B 0,C 180,E1 -22965.728,E2 -22965.728} C_VEL
LIN {X 0,Y 182.266,Z 360.177,A -85,B 0,C 180,E1 -22967.601,E2 -22967.601} C_VEL
LIN {X 0,Y 175.844,Z 349.397,A -85,B 0,C 180,E1 -22969.701,E2 -22969.701} C_VEL
LIN {X 0,Y 173.365,Z 345.597,A -85,B 0,C 180,E1 -22970.547,E2 -22970.547} C_VEL
LIN {X 0,Y 171.734,Z 342.852,A -85,B 0,C 180,E1 -22971.179,E2 -22971.179} C_VEL
LIN {X 0,Y 171.462,Z 341.745,A -85,B 0,C 180,E1 -22971.727,E2 -22971.727} C_VEL
LIN {X 0,Y 171.415,Z 341.621,A -85,B 0,C 180,E1 -22976.808,E2 -22976.808} C_VEL
LIN {X 0,Y 171.458,Z 341.625,A -85,B 0,C 180,E1 -22980.595,E2 -22980.595} C_VEL
LIN {X 0,Y 171.408,Z 341.61,A -85,B 0,C 180,E1 -22985.032,E2 -22985.032} C_VEL
LIN {X 0,Y 171.382,Z 341.632,A -85,B 0,C 180,E1 -22988.817,E2 -22988.817} C_VEL
LIN {X 0,Y 171.333,Z 341.631,A -85,B 0,C 180,E1 -22994.214,E2 -22994.214} C_VEL
LIN {X 0,Y 171.341,Z 341.608,A -85,B 0,C 180,E1 -22998.982,E2 -22998.982} C_VEL
LIN {X 0,Y 171.389,Z 341.603,A -85,B 0,C 180,E1 -23002.041,E2 -23002.041} C_VEL
LIN {X 0,Y 171.4,Z 341.634,A -85,B 0,C 180,E1 -23005.092,E2 -23005.092} C_VEL
LIN {X 0,Y 171.41,Z 341.583,A -85,B 0,C 180,E1 -23010.527,E2 -23010.527} C_VEL
LIN {X 0,Y 171.443,Z 341.628,A -85,B 0,C 180,E1 -23015.799,E2 -23015.799} C_VEL
LIN {X 0,Y 171.521,Z 341.567,A -85,B 0,C 180,E1 -23020.864,E2 -23020.864} C_VEL
LIN {X 0,Y 171.563,Z 341.6,A -85,B 0,C 180,E1 -23025.771,E2 -23025.771} C_VEL
LIN {X 0,Y 171.845,Z 341.552,A -85,B 0,C 180,E1 -23030.584,E2 -23030.584} C_VEL
LIN {X 0,Y 171.786,Z 341.54,A -85,B 0,C 180,E1 -23035.306,E2 -23035.306} C_VEL
LIN {X 0,Y 172.312,Z 341.518,A -85,B 0,C 180,E1 -23039.999,E2 -23039.999} C_VEL
LIN {X 0,Y 171.787,Z 341.537,A -85,B 0,C 180,E1 -23044.693,E2 -23044.693} C_VEL
LIN {X 0,Y 171.848,Z 341.576,A -85,B 0,C 180,E1 -23049.415,E2 -23049.415} C_VEL
LIN {X 0,Y 171.542,Z 341.578,A -85,B 0,C 180,E1 -23054.229,E2 -23054.229} C_VEL
LIN {X 0,Y 171.48,Z 341.625,A -85,B 0,C 180,E1 -23059.499,E2 -23059.499} C_VEL
LIN {X 0,Y 171.444,Z 341.606,A -85,B 0,C 180,E1 -23065.598,E2 -23065.598} C_VEL
LIN {X 0,Y 171.417,Z 341.609,A -85,B 0,C 180,E1 -23070.572,E2 -23070.572} C_VEL
LIN {X 0,Y 171.391,Z 341.634,A -85,B 0,C 180,E1 -23075.034,E2 -23075.034} C_VEL
LIN {X 0,Y 171.342,Z 341.63,A -85,B 0,C 180,E1 -23078.8,E2 -23078.8} C_VEL
LIN {X 0,Y 171.333,Z 341.813,A -85,B 0,C 180,E1 -23084.085,E2 -23084.085} C_VEL
LIN {X 0,Y 171.556,Z 342.753,A -85,B 0,C 180,E1 -23084.579,E2 -23084.579} C_VEL
LIN {X 0,Y 173.469,Z 346.008,A -85,B 0,C 180,E1 -23085.327,E2 -23085.327} C_VEL
LIN {X 0,Y 180.749,Z 359.76,A -85,B 0,C 180,E1 -23087.859,E2 -23087.859} C_VEL
LIN {X 0,Y 186.939,Z 373.326,A -85,B 0,C 180,E1 -23089.89,E2 -23089.89} C_VEL
LIN {X 0,Y 192.87,Z 388.577,A -85,B 0,C 180,E1 -23091.802,E2 -23091.802} C_VEL
LIN {X 0,Y 194.51,Z 393.497,A -85,B 0,C 180,E1 -23092.336,E2 -23092.336} C_VEL
LIN {X 0,Y 195.049,Z 398.76,A -85,B 0,C 180,E1 -23092.674,E2 -23092.674} C_VEL
LIN {X 0,Y 192.227,Z 449.12,A -85,B 0,C 180,E1 -23094.521,E2 -23094.521} C_VEL
LIN {X 0,Y 191.397,Z 458.597,A -85,B 0,C 180,E1 -23095.068,E2 -23095.068} C_VEL
LIN {X 0,Y 190.056,Z 468.381,A -85,B 0,C 180,E1 -23095.832,E2 -23095.832} C_VEL
LIN {X 0,Y 188.098,Z 479.223,A -85,B 0,C 180,E1 -23096.979,E2 -23096.979} C_VEL
LIN {X 0,Y 186.437,Z 484.812,A -85,B 0,C 180,E1 -23097.616,E2 -23097.616} C_VEL
LIN {X 0,Y 181.857,Z 493.083,A -85,B 0,C 180,E1 -23098.533,E2 -23098.533} C_VEL
LIN {X 0,Y 178.025,Z 499.406,A -85,B 0,C 180,E1 -23099.393,E2 -23099.393} C_VEL
LIN {X 0,Y 175.846,Z 504.079,A -85,B 0,C 180,E1 -23100.259,E2 -23100.259} C_VEL
LIN {X 0,Y 175.384,Z 505.641,A -85,B 0,C 180,E1 -23100.6,E2 -23100.6} C_VEL
LIN {X 0,Y 172.3,Z 515.738,A -85,B 0,C 180,E1 -23103.34,E2 -23103.34} C_VEL
LIN {X 0,Y 169.703,Z 524.015,A -85,B 0,C 180,E1 -23106.185,E2 -23106.185} C_VEL
LIN {X 0,Y 167.388,Z 530.885,A -85,B 0,C 180,E1 -23109.091,E2 -23109.091} C_VEL
LIN {X 0,Y 165.852,Z 535.614,A -85,B 0,C 180,E1 -23111.469,E2 -23111.469} C_VEL
LIN {X 0,Y 163.97,Z 541.386,A -85,B 0,C 180,E1 -23115.098,E2 -23115.098} C_VEL
LIN {X 0,Y 162.776,Z 545.918,A -85,B 0,C 180,E1 -23118.796,E2 -23118.796} C_VEL
LIN {X 0,Y 162.042,Z 549.342,A -85,B 0,C 180,E1 -23122.524,E2 -23122.524} C_VEL
LIN {X 0,Y 161.717,Z 552.249,A -85,B 0,C 180,E1 -23127.509,E2 -23127.509} C_VEL
LIN {X 0,Y 161.77,Z 553.198,A -85,B 0,C 180,E1 -23130,E2 -23130} C_VEL
LIN {X 0,Y 161.798,Z 553.651,A -85,B 0,C 180,E1 -23134.984,E2 -23134.984} C_VEL
LIN {X 0,Y 162.122,Z 553.312,A -85,B 0,C 180,E1 -23137.472,E2 -23137.472} C_VEL
LIN {X 0,Y 163.276,Z 551.496,A -85,B 0,C 180,E1 -23142.428,E2 -23142.428} C_VEL
LIN {X 0,Y 165.451,Z 547.916,A -85,B 0,C 180,E1 -23147.298,E2 -23147.298} C_VEL
LIN {X 0,Y 167.976,Z 544.133,A -85,B 0,C 180,E1 -23150.832,E2 -23150.832} C_VEL
LIN {X 0,Y 171.064,Z 539.244,A -85,B 0,C 180,E1 -23154.257,E2 -23154.257} C_VEL
LIN {X 0,Y 173.901,Z 534.287,A -85,B 0,C 180,E1 -23157.035,E2 -23157.035} C_VEL
LIN {X 0,Y 177.222,Z 528.306,A -85,B 0,C 180,E1 -23159.716,E2 -23159.716} C_VEL
LIN {X 0,Y 181.027,Z 521.141,A -85,B 0,C 180,E1 -23162.263,E2 -23162.263} C_VEL
LIN {X 0,Y 185.201,Z 512.459,A -85,B 0,C 180,E1 -23164.696,E2 -23164.696} C_VEL
LIN {X 0,Y 188.769,Z 504.187,A -85,B 0,C 180,E1 -23166.562,E2 -23166.562} C_VEL
LIN {X 0,Y 192.527,Z 494.133,A -85,B 0,C 180,E1 -23168.357,E2 -23168.357} C_VEL
LIN {X 0,Y 195.483,Z 485.031,A -85,B 0,C 180,E1 -23169.654,E2 -23169.654} C_VEL
LIN {X 0,Y 198.496,Z 473.481,A -85,B 0,C 180,E1 -23170.921,E2 -23170.921} C_VEL
LIN {X 0,Y 200.87,Z 462.204,A -85,B 0,C 180,E1 -23171.807,E2 -23171.807} C_VEL
LIN {X 0,Y 202.479,Z 451.748,A -85,B 0,C 180,E1 -23172.394,E2 -23172.394} C_VEL
LIN {X 0,Y 204.005,Z 433.182,A -85,B 0,C 180,E1 -23173.104,E2 -23173.104} C_VEL
LIN {X 0,Y 205.864,Z 407.891,A -85,B 0,C 180,E1 -23173.934,E2 -23173.934} C_VEL
LIN {X 0,Y 201.852,Z 397.568,A -85,B 0,C 180,E1 -23175.989,E2 -23175.989} C_VEL
LIN {X 0,Y 197.343,Z 388.057,A -85,B 0,C 180,E1 -23178.407,E2 -23178.407} C_VEL
LIN {X 0,Y 192.546,Z 379.272,A -85,B 0,C 180,E1 -23181.256,E2 -23181.256} C_VEL
LIN {X 0,Y 189.698,Z 374.548,A -85,B 0,C 180,E1 -23183.109,E2 -23183.109} C_VEL
LIN {X 0,Y 186.876,Z 370.026,A -85,B 0,C 180,E1 -23185.164,E2 -23185.164} C_VEL
LIN {X 0,Y 183.502,Z 364.986,A -85,B 0,C 180,E1 -23187.901,E2 -23187.901} C_VEL
LIN {X 0,Y 180.845,Z 361.925,A -85,B 0,C 180,E1 -23190.347,E2 -23190.347} C_VEL
LIN {X 0,Y 179.851,Z 360.072,A -85,B 0,C 180,E1 -23191.449,E2 -23191.449} C_VEL
LIN {X 0,Y 177.092,Z 357.729,A -85,B 0,C 180,E1 -23194.66,E2 -23194.66} C_VEL
LIN {X 0,Y 175.73,Z 354.904,A -85,B 0,C 180,E1 -23196.903,E2 -23196.903} C_VEL
LIN {X 0,Y 174.338,Z 354.058,A -85,B 0,C 180,E1 -23199.308,E2 -23199.308} C_VEL
LIN {X 0,Y 172.245,Z 352.14,A -85,B 0,C 180,E1 -23207.506,E2 -23207.506} C_VEL
LIN {X 0,Y 172.526,Z 352.263,A -85,B 0,C 180,E1 -23211.214,E2 -23211.214} C_VEL
LIN {X 0,Y 176.188,Z 354.499,A -85,B 0,C 180,E1 -23219.903,E2 -23219.903} C_VEL
LIN {X 0,Y 177.41,Z 357.453,A -85,B 0,C 180,E1 -23221.916,E2 -23221.916} C_VEL
LIN {X 0,Y 179.568,Z 359.672,A -85,B 0,C 180,E1 -23224.49,E2 -23224.49} C_VEL
LIN {X 0,Y 180.562,Z 360.449,A -85,B 0,C 180,E1 -23225.48,E2 -23225.48} C_VEL
LIN {X 0,Y 182.807,Z 363.962,A -85,B 0,C 180,E1 -23227.715,E2 -23227.715} C_VEL
LIN {X 0,Y 184.191,Z 365.414,A -85,B 0,C 180,E1 -23228.884,E2 -23228.884} C_VEL
LIN {X 0,Y 186.804,Z 369.175,A -85,B 0,C 180,E1 -23230.963,E2 -23230.963} C_VEL
LIN {X 0,Y 188.036,Z 370.839,A -85,B 0,C 180,E1 -23231.863,E2 -23231.863} C_VEL
LIN {X 0,Y 191.417,Z 375.726,A -85,B 0,C 180,E1 -23234.146,E2 -23234.146} C_VEL
LIN {X 0,Y 194.786,Z 380.77,A -85,B 0,C 180,E1 -23236.183,E2 -23236.183} C_VEL
LIN {X 0,Y 199.384,Z 389.209,A -85,B 0,C 180,E1 -23238.763,E2 -23238.763} C_VEL
LIN {X 0,Y 204.51,Z 400.409,A -85,B 0,C 180,E1 -23241.411,E2 -23241.411} C_VEL
LIN {X 0,Y 206.079,Z 404.311,A -85,B 0,C 180,E1 -23242.181,E2 -23242.181} C_VEL
LIN {X 0,Y 202.919,Z 445.208,A -85,B 0,C 180,E1 -23243.571,E2 -23243.571} C_VEL
LIN {X 0,Y 201.632,Z 455.009,A -85,B 0,C 180,E1 -23244.069,E2 -23244.069} C_VEL
LIN {X 0,Y 199.937,Z 464.532,A -85,B 0,C 180,E1 -23244.746,E2 -23244.746} C_VEL
LIN {X 0,Y 197.485,Z 475.206,A -85,B 0,C 180,E1 -23245.777,E2 -23245.777} C_VEL
LIN {X 0,Y 195.006,Z 484.129,A -85,B 0,C 180,E1 -23246.876,E2 -23246.876} C_VEL
LIN {X 0,Y 191.463,Z 494.523,A -85,B 0,C 180,E1 -23248.502,E2 -23248.502} C_VEL
LIN {X 0,Y 188.11,Z 503.237,A -85,B 0,C 180,E1 -23250.234,E2 -23250.234} C_VEL
LIN {X 0,Y 184.534,Z 511.375,A -85,B 0,C 180,E1 -23252.222,E2 -23252.222} C_VEL
LIN {X 0,Y 180.094,Z 520.22,A -85,B 0,C 180,E1 -23254.965,E2 -23254.965} C_VEL
LIN {X 0,Y 176.754,Z 526.343,A -85,B 0,C 180,E1 -23257.323,E2 -23257.323} C_VEL
LIN {X 0,Y 172.968,Z 532.898,A -85,B 0,C 180,E1 -23260.55,E2 -23260.55} C_VEL
LIN {X 0,Y 169.925,Z 537.811,A -85,B 0,C 180,E1 -23263.632,E2 -23263.632} C_VEL
LIN {X 0,Y 167.69,Z 541.3,A -85,B 0,C 180,E1 -23266.354,E2 -23266.354} C_VEL
LIN {X 0,Y 165.128,Z 545.023,A -85,B 0,C 180,E1 -23270.327,E2 -23270.327} C_VEL
LIN {X 0,Y 163.098,Z 547.745,A -85,B 0,C 180,E1 -23274.958,E2 -23274.958} C_VEL
LIN {X 0,Y 162.02,Z 548.93,A -85,B 0,C 180,E1 -23278.633,E2 -23278.633} C_VEL
LIN {X 0,Y 161.512,Z 549.266,A -85,B 0,C 180,E1 -23281.403,E2 -23281.403} C_VEL
LIN {X 0,Y 161.244,Z 548.372,A -85,B 0,C 180,E1 -23286.904,E2 -23286.904} C_VEL
LIN {X 0,Y 161.364,Z 547.307,A -85,B 0,C 180,E1 -23289.609,E2 -23289.609} C_VEL
LIN {X 0,Y 161.872,Z 545.289,A -85,B 0,C 180,E1 -23292.782,E2 -23292.782} C_VEL
LIN {X 0,Y 163.083,Z 541.029,A -85,B 0,C 180,E1 -23297.557,E2 -23297.557} C_VEL
LIN {X 0,Y 164.551,Z 536.069,A -85,B 0,C 180,E1 -23301.445,E2 -23301.445} C_VEL
LIN {X 0,Y 166.56,Z 529.856,A -85,B 0,C 180,E1 -23305.159,E2 -23305.159} C_VEL
LIN {X 0,Y 168.971,Z 522.769,A -85,B 0,C 180,E1 -23308.484,E2 -23308.484} C_VEL
LIN {X 0,Y 171.316,Z 515.683,A -85,B 0,C 180,E1 -23311.176,E2 -23311.176} C_VEL
LIN {X 0,Y 173.898,Z 507.285,A -85,B 0,C 180,E1 -23313.766,E2 -23313.766} C_VEL
LIN {X 0,Y 176.697,Z 497.84,A -85,B 0,C 180,E1 -23316.085,E2 -23316.085} C_VEL
LIN {X 0,Y 179.093,Z 488.706,A -85,B 0,C 180,E1 -23317.895,E2 -23317.895} C_VEL
LIN {X 0,Y 180.943,Z 480.654,A -85,B 0,C 180,E1 -23319.22,E2 -23319.22} C_VEL
LIN {X 0,Y 183.116,Z 469.501,A -85,B 0,C 180,E1 -23320.644,E2 -23320.644} C_VEL
LIN {X 0,Y 184.729,Z 458.28,A -85,B 0,C 180,E1 -23321.73,E2 -23321.73} C_VEL
LIN {X 0,Y 185.989,Z 448.083,A -85,B 0,C 180,E1 -23322.411,E2 -23322.411} C_VEL
LIN {X 0,Y 187.271,Z 429.612,A -85,B 0,C 180,E1 -23323.176,E2 -23323.176} C_VEL
LIN {X 0,Y 189.289,Z 392.785,A -85,B 0,C 180,E1 -23324.525,E2 -23324.525} C_VEL
LIN {X 0,Y 182.935,Z 376.064,A -85,B 0,C 180,E1 -23326.653,E2 -23326.653} C_VEL
LIN {X 0,Y 177.17,Z 363.991,A -85,B 0,C 180,E1 -23328.593,E2 -23328.593} C_VEL
LIN {X 0,Y 169.49,Z 351.17,A -85,B 0,C 180,E1 -23331.26,E2 -23331.26} C_VEL
LIN {X 0,Y 167.178,Z 347.665,A -85,B 0,C 180,E1 -23332.102,E2 -23332.102} C_VEL
LIN {X 0,Y 164.932,Z 344.379,A -85,B 0,C 180,E1 -23332.955,E2 -23332.955} C_VEL
LIN {X 0,Y 164.46,Z 342.934,A -85,B 0,C 180,E1 -23333.451,E2 -23333.451} C_VEL
LIN {X 0,Y 164.41,Z 342.535,A -85,B 0,C 180,E1 -23333.96,E2 -23333.96} C_VEL
LIN {X 0,Y 164.341,Z 342.495,A -85,B 0,C 180,E1 -23338.061,E2 -23338.061} C_VEL
LIN {X 0,Y 164.389,Z 342.509,A -85,B 0,C 180,E1 -23341.235,E2 -23341.235} C_VEL
LIN {X 0,Y 164.315,Z 342.51,A -85,B 0,C 180,E1 -23346.784,E2 -23346.784} C_VEL
LIN {X 0,Y 164.302,Z 342.497,A -85,B 0,C 180,E1 -23349.913,E2 -23349.913} C_VEL
LIN {X 0,Y 164.281,Z 342.497,A -85,B 0,C 180,E1 -23353.342,E2 -23353.342} C_VEL
LIN {X 0,Y 164.294,Z 342.516,A -85,B 0,C 180,E1 -23356.809,E2 -23356.809} C_VEL
LIN {X 0,Y 164.298,Z 342.478,A -85,B 0,C 180,E1 -23360.352,E2 -23360.352} C_VEL
LIN {X 0,Y 164.332,Z 342.511,A -85,B 0,C 180,E1 -23364.349,E2 -23364.349} C_VEL
LIN {X 0,Y 164.372,Z 342.466,A -85,B 0,C 180,E1 -23369.13,E2 -23369.13} C_VEL
LIN {X 0,Y 164.397,Z 342.499,A -85,B 0,C 180,E1 -23374.69,E2 -23374.69} C_VEL
LIN {X 0,Y 164.422,Z 342.457,A -85,B 0,C 180,E1 -23380.113,E2 -23380.113} C_VEL
LIN {X 0,Y 164.491,Z 342.47,A -85,B 0,C 180,E1 -23385.146,E2 -23385.146} C_VEL
LIN {X 0,Y 164.766,Z 342.439,A -85,B 0,C 180,E1 -23390.176,E2 -23390.176} C_VEL
LIN {X 0,Y 164.822,Z 342.4,A -85,B 0,C 180,E1 -23392.65,E2 -23392.65} C_VEL
LIN {X 0,Y 165.277,Z 342.394,A -85,B 0,C 180,E1 -23399.999,E2 -23399.999} C_VEL
LIN {X 0,Y 164.825,Z 342.423,A -85,B 0,C 180,E1 -23407.349,E2 -23407.349} C_VEL
LIN {X 0,Y 164.703,Z 342.466,A -85,B 0,C 180,E1 -23411.058,E2 -23411.058} C_VEL
LIN {X 0,Y 164.427,Z 342.479,A -85,B 0,C 180,E1 -23417.409,E2 -23417.409} C_VEL
LIN {X 0,Y 164.42,Z 342.505,A -85,B 0,C 180,E1 -23419.995,E2 -23419.995} C_VEL
LIN {X 0,Y 164.371,Z 342.493,A -85,B 0,C 180,E1 -23426.116,E2 -23426.116} C_VEL
LIN {X 0,Y 164.353,Z 342.488,A -85,B 0,C 180,E1 -23431.214,E2 -23431.214} C_VEL
LIN {X 0,Y 164.279,Z 342.504,A -85,B 0,C 180,E1 -23436.793,E2 -23436.793} C_VEL
LIN {X 0,Y 164.305,Z 342.668,A -85,B 0,C 180,E1 -23442.145,E2 -23442.145} C_VEL
LIN {X 0,Y 164.546,Z 343.728,A -85,B 0,C 180,E1 -23442.69,E2 -23442.69} C_VEL
LIN {X 0,Y 166.08,Z 346.459,A -85,B 0,C 180,E1 -23443.339,E2 -23443.339} C_VEL
LIN {X 0,Y 167.289,Z 348.149,A -85,B 0,C 180,E1 -23443.783,E2 -23443.783} C_VEL
LIN {X 0,Y 170.704,Z 354.016,A -85,B 0,C 180,E1 -23445.051,E2 -23445.051} C_VEL
LIN {X 0,Y 177.436,Z 367.163,A -85,B 0,C 180,E1 -23447.465,E2 -23447.465} C_VEL
LIN {X 0,Y 183.802,Z 382.309,A -85,B 0,C 180,E1 -23449.671,E2 -23449.671} C_VEL
LIN {X 0,Y 188.718,Z 396.019,A -85,B 0,C 180,E1 -23451.343,E2 -23451.343} C_VEL
LIN {X 0,Y 189.04,Z 399.278,A -85,B 0,C 180,E1 -23451.561,E2 -23451.561} C_VEL
LIN {X 0,Y 186.131,Z 448.944,A -85,B 0,C 180,E1 -23453.425,E2 -23453.425} C_VEL
LIN {X 0,Y 185.273,Z 458.45,A -85,B 0,C 180,E1 -23453.987,E2 -23453.987} C_VEL
LIN {X 0,Y 183.773,Z 468.845,A -85,B 0,C 180,E1 -23454.828,E2 -23454.828} C_VEL
LIN {X 0,Y 181.771,Z 479.434,A -85,B 0,C 180,E1 -23455.985,E2 -23455.985} C_VEL
LIN {X 0,Y 179.648,Z 489.551,A -85,B 0,C 180,E1 -23457.458,E2 -23457.458} C_VEL
LIN {X 0,Y 177.016,Z 499.462,A -85,B 0,C 180,E1 -23459.258,E2 -23459.258} C_VEL
LIN {X 0,Y 175.384,Z 505.641,A -85,B 0,C 180,E1 -23460.6,E2 -23460.6} C_VEL
LIN {X 0,Y 173.575,Z 510.237,A -85,B 0,C 180,E1 -23461.65,E2 -23461.65} C_VEL
LIN {X 0,Y 168.783,Z 517.169,A -85,B 0,C 180,E1 -23463.379,E2 -23463.379} C_VEL
LIN {X 0,Y 163.839,Z 523.669,A -85,B 0,C 180,E1 -23465.377,E2 -23465.377} C_VEL
LIN {X 0,Y 161.828,Z 527.314,A -85,B 0,C 180,E1 -23466.831,E2 -23466.831} C_VEL
LIN {X 0,Y 159.083,Z 535.062,A -85,B 0,C 180,E1 -23470.65,E2 -23470.65} C_VEL
LIN {X 0,Y 157.068,Z 540.948,A -85,B 0,C 180,E1 -23474.426,E2 -23474.426} C_VEL
LIN {X 0,Y 155.806,Z 545.566,A -85,B 0,C 180,E1 -23478.288,E2 -23478.288} C_VEL
LIN {X 0,Y 154.99,Z 549.054,A -85,B 0,C 180,E1 -23482.181,E2 -23482.181} C_VEL
LIN {X 0,Y 154.629,Z 552.052,A -85,B 0,C 180,E1 -23487.395,E2 -23487.395} C_VEL
LIN {X 0,Y 154.646,Z 553.253,A -85,B 0,C 180,E1 -23491.172,E2 -23491.172} C_VEL
LIN {X 0,Y 154.721,Z 553.585,A -85,B 0,C 180,E1 -23495.212,E2 -23495.212} C_VEL
LIN {X 0,Y 155.057,Z 553.245,A -85,B 0,C 180,E1 -23497.815,E2 -23497.815} C_VEL
LIN {X 0,Y 156.334,Z 551.536,A -85,B 0,C 180,E1 -23502.989,E2 -23502.989} C_VEL
LIN {X 0,Y 158.662,Z 548.056,A -85,B 0,C 180,E1 -23508.063,E2 -23508.063} C_VEL
LIN {X 0,Y 161.357,Z 544.348,A -85,B 0,C 180,E1 -23511.729,E2 -23511.729} C_VEL
LIN {X 0,Y 164.6,Z 539.555,A -85,B 0,C 180,E1 -23515.275,E2 -23515.275} C_VEL
LIN {X 0,Y 168.235,Z 533.574,A -85,B 0,C 180,E1 -23518.687,E2 -23518.687} C_VEL
LIN {X 0,Y 171.897,Z 527.443,A -85,B 0,C 180,E1 -23521.418,E2 -23521.418} C_VEL
LIN {X 0,Y 175.908,Z 520.132,A -85,B 0,C 180,E1 -23524.01,E2 -23524.01} C_VEL
LIN {X 0,Y 180.309,Z 511.271,A -85,B 0,C 180,E1 -23526.47,E2 -23526.47} C_VEL
LIN {X 0,Y 184.124,Z 502.77,A -85,B 0,C 180,E1 -23528.335,E2 -23528.335} C_VEL
LIN {X 0,Y 187.569,Z 493.903,A -85,B 0,C 180,E1 -23529.915,E2 -23529.915} C_VEL
LIN {X 0,Y 190.645,Z 484.77,A -85,B 0,C 180,E1 -23531.22,E2 -23531.22} C_VEL
LIN {X 0,Y 193.805,Z 473.169,A -85,B 0,C 180,E1 -23532.485,E2 -23532.485} C_VEL
LIN {X 0,Y 196.164,Z 462.482,A -85,B 0,C 180,E1 -23533.331,E2 -23533.331} C_VEL
LIN {X 0,Y 197.963,Z 450.969,A -85,B 0,C 180,E1 -23533.977,E2 -23533.977} C_VEL
LIN {X 0,Y 199.509,Z 433.151,A -85,B 0,C 180,E1 -23534.659,E2 -23534.659} C_VEL
LIN {X 0,Y 201.229,Z 410.213,A -85,B 0,C 180,E1 -23535.437,E2 -23535.437} C_VEL
LIN {X 0,Y 197.379,Z 400.321,A -85,B 0,C 180,E1 -23537.57,E2 -23537.57} C_VEL
LIN {X 0,Y 192.909,Z 390.831,A -85,B 0,C 180,E1 -23540.207,E2 -23540.207} C_VEL
LIN {X 0,Y 187.962,Z 381.59,A -85,B 0,C 180,E1 -23543.488,E2 -23543.488} C_VEL
LIN {X 0,Y 184.374,Z 375.783,A -85,B 0,C 180,E1 -23546.219,E2 -23546.219} C_VEL
LIN {X 0,Y 181.569,Z 371.448,A -85,B 0,C 180,E1 -23548.66,E2 -23548.66} C_VEL
LIN {X 0,Y 178.968,Z 368.198,A -85,B 0,C 180,E1 -23551.221,E2 -23551.221} C_VEL
LIN {X 0,Y 178.07,Z 366.707,A -85,B 0,C 180,E1 -23552.252,E2 -23552.252} C_VEL
LIN {X 0,Y 175.408,Z 364.024,A -85,B 0,C 180,E1 -23555.654,E2 -23555.654} C_VEL
LIN {X 0,Y 174.228,Z 361.506,A -85,B 0,C 180,E1 -23557.77,E2 -23557.77} C_VEL
LIN {X 0,Y 171.311,Z 359.195,A -85,B 0,C 180,E1 -23567.436,E2 -23567.436} C_VEL
LIN {X 0,Y 171.572,Z 359.294,A -85,B 0,C 180,E1 -23571.164,E2 -23571.164} C_VEL
LIN {X 0,Y 174.832,Z 361.51,A -85,B 0,C 180,E1 -23579.367,E2 -23579.367} C_VEL
LIN {X 0,Y 176.268,Z 364.633,A -85,B 0,C 180,E1 -23581.75,E2 -23581.75} C_VEL
LIN {X 0,Y 178.922,Z 367.184,A -85,B 0,C 180,E1 -23584.859,E2 -23584.859} C_VEL
LIN {X 0,Y 181.146,Z 370.643,A -85,B 0,C 180,E1 -23587.165,E2 -23587.165} C_VEL
LIN {X 0,Y 182.398,Z 372.184,A -85,B 0,C 180,E1 -23588.299,E2 -23588.299} C_VEL
LIN {X 0,Y 185.131,Z 375.987,A -85,B 0,C 180,E1 -23590.542,E2 -23590.542} C_VEL
LIN {X 0,Y 189.501,Z 382.676,A -85,B 0,C 180,E1 -23593.7,E2 -23593.7} C_VEL
LIN {X 0,Y 192.357,Z 387.18,A -85,B 0,C 180,E1 -23595.501,E2 -23595.501} C_VEL
LIN {X 0,Y 196.782,Z 395.924,A -85,B 0,C 180,E1 -23598.141,E2 -23598.141} C_VEL
LIN {X 0,Y 201.333,Z 406.471,A -85,B 0,C 180,E1 -23600.619,E2 -23600.619} C_VEL
LIN {X 0,Y 201.417,Z 408.269,A -85,B 0,C 180,E1 -23600.762,E2 -23600.762} C_VEL
LIN {X 0,Y 198.322,Z 445.582,A -85,B 0,C 180,E1 -23602.031,E2 -23602.031} C_VEL
LIN {X 0,Y 196.982,Z 455.313,A -85,B 0,C 180,E1 -23602.534,E2 -23602.534} C_VEL
LIN {X 0,Y 195.437,Z 463.718,A -85,B 0,C 180,E1 -23603.114,E2 -23603.114} C_VEL
LIN {X 0,Y 192.693,Z 475.317,A -85,B 0,C 180,E1 -23604.243,E2 -23604.243} C_VEL
LIN {X 0,Y 189.773,Z 485.178,A -85,B 0,C 180,E1 -23605.485,E2 -23605.485} C_VEL
LIN {X 0,Y 186.24,Z 495.034,A -85,B 0,C 180,E1 -23607.059,E2 -23607.059} C_VEL
LIN {X 0,Y 182.6,Z 503.98,A -85,B 0,C 180,E1 -23608.883,E2 -23608.883} C_VEL
LIN {X 0,Y 179.339,Z 511.088,A -85,B 0,C 180,E1 -23610.628,E2 -23610.628} C_VEL
LIN {X 0,Y 174.766,Z 519.81,A -85,B 0,C 180,E1 -23613.342,E2 -23613.342} C_VEL
LIN {X 0,Y 171.153,Z 526.154,A -85,B 0,C 180,E1 -23615.808,E2 -23615.808} C_VEL
LIN {X 0,Y 166.984,Z 532.84,A -85,B 0,C 180,E1 -23619.148,E2 -23619.148} C_VEL
LIN {X 0,Y 164.435,Z 536.803,A -85,B 0,C 180,E1 -23621.587,E2 -23621.587} C_VEL
LIN {X 0,Y 160.893,Z 541.814,A -85,B 0,C 180,E1 -23625.662,E2 -23625.662} C_VEL
LIN {X 0,Y 158.784,Z 544.702,A -85,B 0,C 180,E1 -23628.803,E2 -23628.803} C_VEL
LIN {X 0,Y 156.206,Z 547.855,A -85,B 0,C 180,E1 -23634.205,E2 -23634.205} C_VEL
LIN {X 0,Y 155.283,Z 548.892,A -85,B 0,C 180,E1 -23637.105,E2 -23637.105} C_VEL
LIN {X 0,Y 154.656,Z 549.262,A -85,B 0,C 180,E1 -23640.009,E2 -23640.009} C_VEL
LIN {X 0,Y 154.137,Z 548.801,A -85,B 0,C 180,E1 -23645.773,E2 -23645.773} C_VEL
LIN {X 0,Y 154.177,Z 547.745,A -85,B 0,C 180,E1 -23648.613,E2 -23648.613} C_VEL
LIN {X 0,Y 154.726,Z 545.575,A -85,B 0,C 180,E1 -23652.53,E2 -23652.53} C_VEL
LIN {X 0,Y 155.394,Z 543.169,A -85,B 0,C 180,E1 -23655.597,E2 -23655.597} C_VEL
LIN {X 0,Y 156.637,Z 538.947,A -85,B 0,C 180,E1 -23659.661,E2 -23659.661} C_VEL
LIN {X 0,Y 158.116,Z 534.478,A -85,B 0,C 180,E1 -23662.979,E2 -23662.979} C_VEL
LIN {X 0,Y 159.575,Z 530.273,A -85,B 0,C 180,E1 -23665.58,E2 -23665.58} C_VEL
LIN {X 0,Y 161.693,Z 524.295,A -85,B 0,C 180,E1 -23668.606,E2 -23668.606} C_VEL
LIN {X 0,Y 164.495,Z 516.243,A -85,B 0,C 180,E1 -23671.837,E2 -23671.837} C_VEL
LIN {X 0,Y 167.171,Z 507.935,A -85,B 0,C 180,E1 -23674.521,E2 -23674.521} C_VEL
LIN {X 0,Y 169.839,Z 499.494,A -85,B 0,C 180,E1 -23676.718,E2 -23676.718} C_VEL
LIN {X 0,Y 172.557,Z 489.606,A -85,B 0,C 180,E1 -23678.786,E2 -23678.786} C_VEL
LIN {X 0,Y 174.866,Z 479.823,A -85,B 0,C 180,E1 -23680.42,E2 -23680.42} C_VEL
LIN {X 0,Y 176.933,Z 469.638,A -85,B 0,C 180,E1 -23681.746,E2 -23681.746} C_VEL
LIN {X 0,Y 178.624,Z 458.417,A -85,B 0,C 180,E1 -23682.859,E2 -23682.859} C_VEL
LIN {X 0,Y 180.016,Z 447.011,A -85,B 0,C 180,E1 -23683.619,E2 -23683.619} C_VEL
LIN {X 0,Y 181.442,Z 426.773,A -85,B 0,C 180,E1 -23684.451,E2 -23684.451} C_VEL
LIN {X 0,Y 183.28,Z 394.696,A -85,B 0,C 180,E1 -23685.653,E2 -23685.653} C_VEL
LIN {X 0,Y 177.621,Z 379.499,A -85,B 0,C 180,E1 -23687.671,E2 -23687.671} C_VEL
LIN {X 0,Y 172.277,Z 368.166,A -85,B 0,C 180,E1 -23689.583,E2 -23689.583} C_VEL
LIN {X 0,Y 164.899,Z 355.831,A -85,B 0,C 180,E1 -23692.273,E2 -23692.273} C_VEL
LIN {X 0,Y 160.268,Z 348.603,A -85,B 0,C 180,E1 -23694.114,E2 -23694.114} C_VEL
LIN {X 0,Y 157.935,Z 345.396,A -85,B 0,C 180,E1 -23695.082,E2 -23695.082} C_VEL
LIN {X 0,Y 157.434,Z 343.789,A -85,B 0,C 180,E1 -23695.657,E2 -23695.657} C_VEL
LIN {X 0,Y 157.312,Z 343.378,A -85,B 0,C 180,E1 -23696.681,E2 -23696.681} C_VEL
LIN {X 0,Y 157.285,Z 343.379,A -85,B 0,C 180,E1 -23702.426,E2 -23702.426} C_VEL
LIN {X 0,Y 157.285,Z 343.38,A -85,B 0,C 180,E1 -23706.456,E2 -23706.456} C_VEL
LIN {X 0,Y 157.215,Z 343.369,A -85,B 0,C 180,E1 -23712.11,E2 -23712.11} C_VEL
LIN {X 0,Y 157.213,Z 343.38,A -85,B 0,C 180,E1 -23717.889,E2 -23717.889} C_VEL
LIN {X 0,Y 157.27,Z 343.38,A -85,B 0,C 180,E1 -23723.551,E2 -23723.551} C_VEL
LIN {X 0,Y 157.285,Z 343.36,A -85,B 0,C 180,E1 -23728.102,E2 -23728.102} C_VEL
LIN {X 0,Y 157.311,Z 343.362,A -85,B 0,C 180,E1 -23733.463,E2 -23733.463} C_VEL
LIN {X 0,Y 157.364,Z 343.34,A -85,B 0,C 180,E1 -23739.699,E2 -23739.699} C_VEL
LIN {X 0,Y 157.423,Z 343.337,A -85,B 0,C 180,E1 -23744.462,E2 -23744.462} C_VEL
LIN {X 0,Y 157.689,Z 343.327,A -85,B 0,C 180,E1 -23749.73,E2 -23749.73} C_VEL
LIN {X 0,Y 157.76,Z 343.281,A -85,B 0,C 180,E1 -23752.319,E2 -23752.319} C_VEL
LIN {X 0,Y 158.239,Z 343.271,A -85,B 0,C 180,E1 -23759.999,E2 -23759.999} C_VEL
LIN {X 0,Y 157.763,Z 343.306,A -85,B 0,C 180,E1 -23767.68,E2 -23767.68} C_VEL
LIN {X 0,Y 157.632,Z 343.345,A -85,B 0,C 180,E1 -23771.225,E2 -23771.225} C_VEL
LIN {X 0,Y 157.406,Z 343.336,A -85,B 0,C 180,E1 -23775.538,E2 -23775.538} C_VEL
LIN {X 0,Y 157.311,Z 343.381,A -85,B 0,C 180,E1 -23780.94,E2 -23780.94} C_VEL
LIN {X 0,Y 157.31,Z 343.38,A -85,B 0,C 180,E1 -23786.68,E2 -23786.68} C_VEL
LIN {X 0,Y 157.264,Z 343.375,A -85,B 0,C 180,E1 -23792.429,E2 -23792.429} C_VEL
LIN {X 0,Y 157.258,Z 343.38,A -85,B 0,C 180,E1 -23796.443,E2 -23796.443} C_VEL
LIN {X 0,Y 157.286,Z 343.54,A -85,B 0,C 180,E1 -23799.914,E2 -23799.914} C_VEL
LIN {X 0,Y 157.549,Z 344.823,A -85,B 0,C 180,E1 -23800.562,E2 -23800.562} C_VEL
LIN {X 0,Y 159.231,Z 347.52,A -85,B 0,C 180,E1 -23801.312,E2 -23801.312} C_VEL
LIN {X 0,Y 160.145,Z 348.709,A -85,B 0,C 180,E1 -23801.681,E2 -23801.681} C_VEL
LIN {X 0,Y 165.452,Z 357.358,A -85,B 0,C 180,E1 -23803.802,E2 -23803.802} C_VEL
LIN {X 0,Y 171.637,Z 369.579,A -85,B 0,C 180,E1 -23806.158,E2 -23806.158} C_VEL
LIN {X 0,Y 177.353,Z 382.862,A -85,B 0,C 180,E1 -23808.269,E2 -23808.269} C_VEL
LIN {X 0,Y 182.85,Z 397.831,A -85,B 0,C 180,E1 -23810.238,E2 -23810.238} C_VEL
LIN {X 0,Y 182.896,Z 402.495,A -85,B 0,C 180,E1 -23810.477,E2 -23810.477} C_VEL
LIN {X 0,Y 180.107,Z 448.582,A -85,B 0,C 180,E1 -23812.255,E2 -23812.255} C_VEL
LIN {X 0,Y 179.203,Z 458.175,A -85,B 0,C 180,E1 -23812.828,E2 -23812.828} C_VEL
LIN {X 0,Y 177.765,Z 468.015,A -85,B 0,C 180,E1 -23813.627,E2 -23813.627} C_VEL
LIN {X 0,Y 175.569,Z 479.221,A -85,B 0,C 180,E1 -23814.87,E2 -23814.87} C_VEL
LIN {X 0,Y 173.269,Z 489.746,A -85,B 0,C 180,E1 -23816.451,E2 -23816.451} C_VEL
LIN {X 0,Y 170.951,Z 498.371,A -85,B 0,C 180,E1 -23818.041,E2 -23818.041} C_VEL
LIN {X 0,Y 168.106,Z 507.849,A -85,B 0,C 180,E1 -23820.234,E2 -23820.234} C_VEL
LIN {X 0,Y 165.365,Z 516.676,A -85,B 0,C 180,E1 -23822.815,E2 -23822.815} C_VEL
LIN {X 0,Y 163.122,Z 523.335,A -85,B 0,C 180,E1 -23825.161,E2 -23825.161} C_VEL
LIN {X 0,Y 161.828,Z 527.314,A -85,B 0,C 180,E1 -23826.831,E2 -23826.831} C_VEL
LIN {X 0,Y 159.884,Z 530.879,A -85,B 0,C 180,E1 -23828.365,E2 -23828.365} C_VEL
LIN {X 0,Y 155.217,Z 536.056,A -85,B 0,C 180,E1 -23830.934,E2 -23830.934} C_VEL
LIN {X 0,Y 150.84,Z 540.583,A -85,B 0,C 180,E1 -23833.82,E2 -23833.82} C_VEL
LIN {X 0,Y 149.403,Z 542.979,A -85,B 0,C 180,E1 -23835.801,E2 -23835.801} C_VEL
LIN {X 0,Y 148.488,Z 546.409,A -85,B 0,C 180,E1 -23839.087,E2 -23839.087} C_VEL
LIN {X 0,Y 147.959,Z 548.733,A -85,B 0,C 180,E1 -23841.807,E2 -23841.807} C_VEL
LIN {X 0,Y 147.527,Z 551.85,A -85,B 0,C 180,E1 -23847.269,E2 -23847.269} C_VEL
LIN {X 0,Y 147.586,Z 552.808,A -85,B 0,C 180,E1 -23850,E2 -23850} C_VEL
LIN {X 0,Y 147.646,Z 553.515,A -85,B 0,C 180,E1 -23855.463,E2 -23855.463} C_VEL
LIN {X 0,Y 148.551,Z 552.532,A -85,B 0,C 180,E1 -23860.908,E2 -23860.908} C_VEL
LIN {X 0,Y 149.417,Z 551.554,A -85,B 0,C 180,E1 -23863.602,E2 -23863.602} C_VEL
LIN {X 0,Y 151.906,Z 548.214,A -85,B 0,C 180,E1 -23868.896,E2 -23868.896} C_VEL
LIN {X 0,Y 154.771,Z 544.598,A -85,B 0,C 180,E1 -23872.704,E2 -23872.704} C_VEL
LIN {X 0,Y 158.194,Z 539.894,A -85,B 0,C 180,E1 -23876.376,E2 -23876.376} C_VEL
LIN {X 0,Y 161.855,Z 534.344,A -85,B 0,C 180,E1 -23879.725,E2 -23879.725} C_VEL
LIN {X 0,Y 165.918,Z 527.987,A -85,B 0,C 180,E1 -23882.688,E2 -23882.688} C_VEL
LIN {X 0,Y 170.11,Z 520.804,A -85,B 0,C 180,E1 -23885.338,E2 -23885.338} C_VEL
LIN {X 0,Y 174.697,Z 512.111,A -85,B 0,C 180,E1 -23887.843,E2 -23887.843} C_VEL
LIN {X 0,Y 179.172,Z 502.613,A -85,B 0,C 180,E1 -23889.964,E2 -23889.964} C_VEL
LIN {X 0,Y 182.747,Z 493.77,A -85,B 0,C 180,E1 -23891.559,E2 -23891.559} C_VEL
LIN {X 0,Y 185.988,Z 484.647,A -85,B 0,C 180,E1 -23892.857,E2 -23892.857} C_VEL
LIN {X 0,Y 189.272,Z 473.08,A -85,B 0,C 180,E1 -23894.124,E2 -23894.124} C_VEL
LIN {X 0,Y 191.716,Z 462.373,A -85,B 0,C 180,E1 -23894.971,E2 -23894.971} C_VEL
LIN {X 0,Y 193.559,Z 451.085,A -85,B 0,C 180,E1 -23895.605,E2 -23895.605} C_VEL
LIN {X 0,Y 195.239,Z 432.663,A -85,B 0,C 180,E1 -23896.307,E2 -23896.307} C_VEL
LIN {X 0,Y 196.772,Z 412.703,A -85,B 0,C 180,E1 -23897,E2 -23897} C_VEL
LIN {X 0,Y 193.259,Z 403.603,A -85,B 0,C 180,E1 -23899.113,E2 -23899.113} C_VEL
LIN {X 0,Y 189.461,Z 395.301,A -85,B 0,C 180,E1 -23901.564,E2 -23901.564} C_VEL
LIN {X 0,Y 185.155,Z 386.999,A -85,B 0,C 180,E1 -23904.671,E2 -23904.671} C_VEL
LIN {X 0,Y 181.73,Z 381.17,A -85,B 0,C 180,E1 -23907.486,E2 -23907.486} C_VEL
LIN {X 0,Y 179.671,Z 377.899,A -85,B 0,C 180,E1 -23909.436,E2 -23909.436} C_VEL
LIN {X 0,Y 177.07,Z 374.358,A -85,B 0,C 180,E1 -23912.182,E2 -23912.182} C_VEL
LIN {X 0,Y 176.484,Z 373.415,A -85,B 0,C 180,E1 -23912.906,E2 -23912.906} C_VEL
LIN {X 0,Y 173.852,Z 370.448,A -85,B 0,C 180,E1 -23916.545,E2 -23916.545} C_VEL
LIN {X 0,Y 172.992,Z 368.405,A -85,B 0,C 180,E1 -23918.266,E2 -23918.266} C_VEL
LIN {X 0,Y 170.362,Z 366.15,A -85,B 0,C 180,E1 -23928.097,E2 -23928.097} C_VEL
LIN {X 0,Y 170.723,Z 366.48,A -85,B 0,C 180,E1 -23931.717,E2 -23931.717} C_VEL
LIN {X 0,Y 173.489,Z 368.405,A -85,B 0,C 180,E1 -23938.793,E2 -23938.793} C_VEL
LIN {X 0,Y 175.062,Z 371.64,A -85,B 0,C 180,E1 -23941.469,E2 -23941.469} C_VEL
LIN {X 0,Y 177.264,Z 373.88,A -85,B 0,C 180,E1 -23944.193,E2 -23944.193} C_VEL
LIN {X 0,Y 179.771,Z 377.604,A -85,B 0,C 180,E1 -23946.86,E2 -23946.86} C_VEL
LIN {X 0,Y 183.617,Z 383.361,A -85,B 0,C 180,E1 -23950.265,E2 -23950.265} C_VEL
LIN {X 0,Y 188.05,Z 390.196,A -85,B 0,C 180,E1 -23953.538,E2 -23953.538} C_VEL
LIN {X 0,Y 192.113,Z 398.003,A -85,B 0,C 180,E1 -23956.194,E2 -23956.194} C_VEL
LIN {X 0,Y 196.303,Z 407.682,A -85,B 0,C 180,E1 -23958.73,E2 -23958.73} C_VEL
LIN {X 0,Y 197.059,Z 409.736,A -85,B 0,C 180,E1 -23959.172,E2 -23959.172} C_VEL
LIN {X 0,Y 193.975,Z 445.498,A -85,B 0,C 180,E1 -23960.393,E2 -23960.393} C_VEL
LIN {X 0,Y 192.572,Z 455.363,A -85,B 0,C 180,E1 -23960.9,E2 -23960.9} C_VEL
LIN {X 0,Y 190.757,Z 464.672,A -85,B 0,C 180,E1 -23961.557,E2 -23961.557} C_VEL
LIN {X 0,Y 188.002,Z 475.745,A -85,B 0,C 180,E1 -23962.649,E2 -23962.649} C_VEL
LIN {X 0,Y 185.247,Z 484.66,A -85,B 0,C 180,E1 -23963.757,E2 -23963.757} C_VEL
LIN {X 0,Y 181.335,Z 495.152,A -85,B 0,C 180,E1 -23965.442,E2 -23965.442} C_VEL
LIN {X 0,Y 177.742,Z 503.613,A -85,B 0,C 180,E1 -23967.17,E2 -23967.17} C_VEL
LIN {X 0,Y 173.905,Z 511.515,A -85,B 0,C 180,E1 -23969.146,E2 -23969.146} C_VEL
LIN {X 0,Y 169.406,Z 519.712,A -85,B 0,C 180,E1 -23971.738,E2 -23971.738} C_VEL
LIN {X 0,Y 165.665,Z 525.961,A -85,B 0,C 180,E1 -23974.183,E2 -23974.183} C_VEL
LIN {X 0,Y 161.128,Z 532.783,A -85,B 0,C 180,E1 -23977.637,E2 -23977.637} C_VEL
LIN {X 0,Y 156.838,Z 538.76,A -85,B 0,C 180,E1 -23981.714,E2 -23981.714} C_VEL
LIN {X 0,Y 154.058,Z 542.413,A -85,B 0,C 180,E1 -23985.001,E2 -23985.001} C_VEL
LIN {X 0,Y 152.277,Z 544.708,A -85,B 0,C 180,E1 -23987.6,E2 -23987.6} C_VEL
LIN {X 0,Y 149.478,Z 547.857,A -85,B 0,C 180,E1 -23993.063,E2 -23993.063} C_VEL
LIN {X 0,Y 148.621,Z 548.68,A -85,B 0,C 180,E1 -23995.427,E2 -23995.427} C_VEL
LIN {X 0,Y 147.73,Z 549.306,A -85,B 0,C 180,E1 -23998.907,E2 -23998.907} C_VEL
LIN {X 0,Y 147.284,Z 549.444,A -85,B 0,C 180,E1 -24001.499,E2 -24001.499} C_VEL
LIN {X 0,Y 147.027,Z 548.957,A -85,B 0,C 180,E1 -24005.261,E2 -24005.261} C_VEL
LIN {X 0,Y 147.246,Z 546.921,A -85,B 0,C 180,E1 -24010.482,E2 -24010.482} C_VEL
LIN {X 0,Y 148.097,Z 544.041,A -85,B 0,C 180,E1 -24014.871,E2 -24014.871} C_VEL
LIN {X 0,Y 149.32,Z 540.047,A -85,B 0,C 180,E1 -24019.149,E2 -24019.149} C_VEL
LIN {X 0,Y 150.412,Z 536.808,A -85,B 0,C 180,E1 -24021.942,E2 -24021.942} C_VEL
LIN {X 0,Y 152.583,Z 530.674,A -85,B 0,C 180,E1 -24026.039,E2 -24026.039} C_VEL
LIN {X 0,Y 154.867,Z 524.496,A -85,B 0,C 180,E1 -24029.308,E2 -24029.308} C_VEL
LIN {X 0,Y 157.695,Z 516.775,A -85,B 0,C 180,E1 -24032.555,E2 -24032.555} C_VEL
LIN {X 0,Y 160.824,Z 507.483,A -85,B 0,C 180,E1 -24035.643,E2 -24035.643} C_VEL
LIN {X 0,Y 163.754,Z 498.44,A -85,B 0,C 180,E1 -24038.018,E2 -24038.018} C_VEL
LIN {X 0,Y 166.445,Z 488.911,A -85,B 0,C 180,E1 -24040.031,E2 -24040.031} C_VEL
LIN {X 0,Y 168.473,Z 480.845,A -85,B 0,C 180,E1 -24041.429,E2 -24041.429} C_VEL
LIN {X 0,Y 170.805,Z 469.707,A -85,B 0,C 180,E1 -24042.929,E2 -24042.929} C_VEL
LIN {X 0,Y 172.579,Z 458.464,A -85,B 0,C 180,E1 -24044.068,E2 -24044.068} C_VEL
LIN {X 0,Y 173.957,Z 447.901,A -85,B 0,C 180,E1 -24044.798,E2 -24044.798} C_VEL
LIN {X 0,Y 175.304,Z 430.03,A -85,B 0,C 180,E1 -24045.571,E2 -24045.571} C_VEL
LIN {X 0,Y 177.202,Z 396.201,A -85,B 0,C 180,E1 -24046.898,E2 -24046.898} C_VEL
LIN {X 0,Y 172.52,Z 383.369,A -85,B 0,C 180,E1 -24048.69,E2 -24048.69} C_VEL
LIN {X 0,Y 167.595,Z 372.71,A -85,B 0,C 180,E1 -24050.542,E2 -24050.542} C_VEL
LIN {X 0,Y 160.472,Z 360.584,A -85,B 0,C 180,E1 -24053.303,E2 -24053.303} C_VEL
LIN {X 0,Y 155.18,Z 352.557,A -85,B 0,C 180,E1 -24055.52,E2 -24055.52} C_VEL
LIN {X 0,Y 152.831,Z 348.86,A -85,B 0,C 180,E1 -24056.575,E2 -24056.575} C_VEL
LIN {X 0,Y 151.066,Z 346.824,A -85,B 0,C 180,E1 -24057.349,E2 -24057.349} C_VEL
LIN {X 0,Y 150.387,Z 345.108,A -85,B 0,C 180,E1 -24057.861,E2 -24057.861} C_VEL
LIN {X 0,Y 150.212,Z 344.305,A -85,B 0,C 180,E1 -24058.658,E2 -24058.658} C_VEL
LIN {X 0,Y 150.201,Z 344.25,A -85,B 0,C 180,E1 -24064.159,E2 -24064.159} C_VEL
LIN {X 0,Y 150.213,Z 344.274,A -85,B 0,C 180,E1 -24067.462,E2 -24067.462} C_VEL
LIN {X 0,Y 150.155,Z 344.248,A -85,B 0,C 180,E1 -24071.506,E2 -24071.506} C_VEL
LIN {X 0,Y 150.129,Z 344.284,A -85,B 0,C 180,E1 -24075.396,E2 -24075.396} C_VEL
LIN {X 0,Y 150.152,Z 344.244,A -85,B 0,C 180,E1 -24079.058,E2 -24079.058} C_VEL
LIN {X 0,Y 150.181,Z 344.248,A -85,B 0,C 180,E1 -24082.707,E2 -24082.707} C_VEL
LIN {X 0,Y 150.21,Z 344.251,A -85,B 0,C 180,E1 -24087.372,E2 -24087.372} C_VEL
LIN {X 0,Y 150.24,Z 344.23,A -85,B 0,C 180,E1 -24092.722,E2 -24092.722} C_VEL
LIN {X 0,Y 150.289,Z 344.226,A -85,B 0,C 180,E1 -24099.272,E2 -24099.272} C_VEL
LIN {X 0,Y 150.326,Z 344.21,A -85,B 0,C 180,E1 -24103.709,E2 -24103.709} C_VEL
LIN {X 0,Y 150.609,Z 344.214,A -85,B 0,C 180,E1 -24109.242,E2 -24109.242} C_VEL
LIN {X 0,Y 150.683,Z 344.164,A -85,B 0,C 180,E1 -24111.956,E2 -24111.956} C_VEL
LIN {X 0,Y 151.199,Z 344.147,A -85,B 0,C 180,E1 -24119.999,E2 -24119.999} C_VEL
LIN {X 0,Y 150.702,Z 344.19,A -85,B 0,C 180,E1 -24128.042,E2 -24128.042} C_VEL
LIN {X 0,Y 150.575,Z 344.222,A -85,B 0,C 180,E1 -24131.429,E2 -24131.429} C_VEL
LIN {X 0,Y 150.311,Z 344.223,A -85,B 0,C 180,E1 -24136.292,E2 -24136.292} C_VEL
LIN {X 0,Y 150.285,Z 344.259,A -85,B 0,C 180,E1 -24140.724,E2 -24140.724} C_VEL
LIN {X 0,Y 150.239,Z 344.268,A -85,B 0,C 180,E1 -24147.276,E2 -24147.276} C_VEL
LIN {X 0,Y 150.205,Z 344.255,A -85,B 0,C 180,E1 -24152.625,E2 -24152.625} C_VEL
LIN {X 0,Y 150.198,Z 344.428,A -85,B 0,C 180,E1 -24157.465,E2 -24157.465} C_VEL
LIN {X 0,Y 150.455,Z 345.613,A -85,B 0,C 180,E1 -24158.131,E2 -24158.131} C_VEL
LIN {X 0,Y 152.041,Z 348.259,A -85,B 0,C 180,E1 -24158.928,E2 -24158.928} C_VEL
LIN {X 0,Y 153.196,Z 349.568,A -85,B 0,C 180,E1 -24159.426,E2 -24159.426} C_VEL
LIN {X 0,Y 155.322,Z 352.871,A -85,B 0,C 180,E1 -24160.372,E2 -24160.372} C_VEL
LIN {X 0,Y 160.454,Z 361.01,A -85,B 0,C 180,E1 -24162.544,E2 -24162.544} C_VEL
LIN {X 0,Y 167.195,Z 374.626,A -85,B 0,C 180,E1 -24165.287,E2 -24165.287} C_VEL
LIN {X 0,Y 172.949,Z 388.615,A -85,B 0,C 180,E1 -24167.528,E2 -24167.528} C_VEL
LIN {X 0,Y 177.104,Z 400.207,A -85,B 0,C 180,E1 -24169.113,E2 -24169.113} C_VEL
LIN {X 0,Y 174.176,Z 447.877,A -85,B 0,C 180,E1 -24170.999,E2 -24170.999} C_VEL
LIN {X 0,Y 173.173,Z 458.124,A -85,B 0,C 180,E1 -24171.621,E2 -24171.621} C_VEL
LIN {X 0,Y 171.626,Z 468.279,A -85,B 0,C 180,E1 -24172.473,E2 -24172.473} C_VEL
LIN {X 0,Y 169.338,Z 479.399,A -85,B 0,C 180,E1 -24173.742,E2 -24173.742} C_VEL
LIN {X 0,Y 167.398,Z 488.373,A -85,B 0,C 180,E1 -24175.108,E2 -24175.108} C_VEL
LIN {X 0,Y 164.553,Z 498.459,A -85,B 0,C 180,E1 -24177.006,E2 -24177.006} C_VEL
LIN {X 0,Y 161.586,Z 507.904,A -85,B 0,C 180,E1 -24179.266,E2 -24179.266} C_VEL
LIN {X 0,Y 159.017,Z 515.843,A -85,B 0,C 180,E1 -24181.634,E2 -24181.634} C_VEL
LIN {X 0,Y 156.391,Z 523.297,A -85,B 0,C 180,E1 -24184.348,E2 -24184.348} C_VEL
LIN {X 0,Y 153.65,Z 530.897,A -85,B 0,C 180,E1 -24187.83,E2 -24187.83} C_VEL
LIN {X 0,Y 151.585,Z 536.593,A -85,B 0,C 180,E1 -24191.062,E2 -24191.062} C_VEL
LIN {X 0,Y 149.682,Z 542.1,A -85,B 0,C 180,E1 -24195.034,E2 -24195.034} C_VEL
LIN {X 0,Y 149.403,Z 542.979,A -85,B 0,C 180,E1 -24195.801,E2 -24195.801} C_VEL
LIN {X 0,Y 148.111,Z 545.315,A -85,B 0,C 180,E1 -24197.847,E2 -24197.847} C_VEL
LIN {X 0,Y 144.516,Z 548.377,A -85,B 0,C 180,E1 -24201.254,E2 -24201.254} C_VEL
LIN {X 0,Y 141.73,Z 550.314,A -85,B 0,C 180,E1 -24204.149,E2 -24204.149} C_VEL
LIN {X 0,Y 140.536,Z 551.407,A -85,B 0,C 180,E1 -24206.475,E2 -24206.475} C_VEL
LIN {X 0,Y 140.424,Z 551.696,A -85,B 0,C 180,E1 -24207.274,E2 -24207.274} C_VEL
LIN {X 0,Y 140.5,Z 552.605,A -85,B 0,C 180,E1 -24210,E2 -24210} C_VEL
LIN {X 0,Y 140.569,Z 553.425,A -85,B 0,C 180,E1 -24215.739,E2 -24215.739} C_VEL
LIN {X 0,Y 141.585,Z 552.543,A -85,B 0,C 180,E1 -24221.452,E2 -24221.452} C_VEL
LIN {X 0,Y 142.509,Z 551.566,A -85,B 0,C 180,E1 -24224.275,E2 -24224.275} C_VEL
LIN {X 0,Y 145.187,Z 548.38,A -85,B 0,C 180,E1 -24229.806,E2 -24229.806} C_VEL
LIN {X 0,Y 148.242,Z 544.843,A -85,B 0,C 180,E1 -24233.764,E2 -24233.764} C_VEL
LIN {X 0,Y 151.852,Z 540.23,A -85,B 0,C 180,E1 -24237.569,E2 -24237.569} C_VEL
LIN {X 0,Y 155.985,Z 534.406,A -85,B 0,C 180,E1 -24241.216,E2 -24241.216} C_VEL
LIN {X 0,Y 160.877,Z 527.168,A -85,B 0,C 180,E1 -24244.605,E2 -24244.605} C_VEL
LIN {X 0,Y 165.307,Z 519.869,A -85,B 0,C 180,E1 -24247.289,E2 -24247.289} C_VEL
LIN {X 0,Y 170.163,Z 511.02,A -85,B 0,C 180,E1 -24249.805,E2 -24249.805} C_VEL
LIN {X 0,Y 174.376,Z 502.523,A -85,B 0,C 180,E1 -24251.683,E2 -24251.683} C_VEL
LIN {X 0,Y 178.117,Z 493.678,A -85,B 0,C 180,E1 -24253.28,E2 -24253.28} C_VEL
LIN {X 0,Y 181.491,Z 484.555,A -85,B 0,C 180,E1 -24254.577,E2 -24254.577} C_VEL
LIN {X 0,Y 184.906,Z 472.988,A -85,B 0,C 180,E1 -24255.841,E2 -24255.841} C_VEL
LIN {X 0,Y 187.505,Z 461.986,A -85,B 0,C 180,E1 -24256.697,E2 -24256.697} C_VEL
LIN {X 0,Y 189.346,Z 451.024,A -85,B 0,C 180,E1 -24257.311,E2 -24257.311} C_VEL
LIN {X 0,Y 191.112,Z 432.39,A -85,B 0,C 180,E1 -24258.025,E2 -24258.025} C_VEL
LIN {X 0,Y 192.475,Z 415.21,A -85,B 0,C 180,E1 -24258.637,E2 -24258.637} C_VEL
LIN {X 0,Y 189.044,Z 406.241,A -85,B 0,C 180,E1 -24260.92,E2 -24260.92} C_VEL
LIN {X 0,Y 185.7,Z 399.005,A -85,B 0,C 180,E1 -24263.283,E2 -24263.283} C_VEL
LIN {X 0,Y 182.393,Z 392.358,A -85,B 0,C 180,E1 -24265.918,E2 -24265.918} C_VEL
LIN {X 0,Y 179.795,Z 387.628,A -85,B 0,C 180,E1 -24268.233,E2 -24268.233} C_VEL
LIN {X 0,Y 177.945,Z 384.482,A -85,B 0,C 180,E1 -24270.094,E2 -24270.094} C_VEL
LIN {X 0,Y 175.368,Z 380.773,A -85,B 0,C 180,E1 -24273.001,E2 -24273.001} C_VEL
LIN {X 0,Y 172.26,Z 376.666,A -85,B 0,C 180,E1 -24277.617,E2 -24277.617} C_VEL
LIN {X 0,Y 171.703,Z 375.314,A -85,B 0,C 180,E1 -24278.885,E2 -24278.885} C_VEL
LIN {X 0,Y 169.426,Z 373.184,A -85,B 0,C 180,E1 -24288.03,E2 -24288.03} C_VEL
LIN {X 0,Y 169.771,Z 373.528,A -85,B 0,C 180,E1 -24291.67,E2 -24291.67} C_VEL
LIN {X 0,Y 172.193,Z 375.255,A -85,B 0,C 180,E1 -24298.202,E2 -24298.202} C_VEL
LIN {X 0,Y 173.829,Z 378.612,A -85,B 0,C 180,E1 -24301.138,E2 -24301.138} C_VEL
LIN {X 0,Y 175.695,Z 380.638,A -85,B 0,C 180,E1 -24303.571,E2 -24303.571} C_VEL
LIN {X 0,Y 178.108,Z 384.252,A -85,B 0,C 180,E1 -24306.266,E2 -24306.266} C_VEL
LIN {X 0,Y 181.555,Z 389.748,A -85,B 0,C 180,E1 -24309.514,E2 -24309.514} C_VEL
LIN {X 0,Y 185.678,Z 396.451,A -85,B 0,C 180,E1 -24312.73,E2 -24312.73} C_VEL
LIN {X 0,Y 189.574,Z 404.367,A -85,B 0,C 180,E1 -24315.445,E2 -24315.445} C_VEL
LIN {X 0,Y 192.784,Z 412.469,A -85,B 0,C 180,E1 -24317.554,E2 -24317.554} C_VEL
LIN {X 0,Y 189.816,Z 445.265,A -85,B 0,C 180,E1 -24318.675,E2 -24318.675} C_VEL
LIN {X 0,Y 188.408,Z 455.008,A -85,B 0,C 180,E1 -24319.168,E2 -24319.168} C_VEL
LIN {X 0,Y 186.466,Z 464.604,A -85,B 0,C 180,E1 -24319.829,E2 -24319.829} C_VEL
LIN {X 0,Y 183.786,Z 475.133,A -85,B 0,C 180,E1 -24320.854,E2 -24320.854} C_VEL
LIN {X 0,Y 180.417,Z 485.493,A -85,B 0,C 180,E1 -24322.15,E2 -24322.15} C_VEL
LIN {X 0,Y 176.59,Z 495.319,A -85,B 0,C 180,E1 -24323.743,E2 -24323.743} C_VEL
LIN {X 0,Y 172.479,Z 504.451,A -85,B 0,C 180,E1 -24325.641,E2 -24325.641} C_VEL
LIN {X 0,Y 168.432,Z 512.297,A -85,B 0,C 180,E1 -24327.659,E2 -24327.659} C_VEL
LIN {X 0,Y 164.283,Z 519.52,A -85,B 0,C 180,E1 -24329.97,E2 -24329.97} C_VEL
LIN {X 0,Y 159.355,Z 527.11,A -85,B 0,C 180,E1 -24333.076,E2 -24333.076} C_VEL
LIN {X 0,Y 155.44,Z 532.708,A -85,B 0,C 180,E1 -24336,E2 -24336} C_VEL
LIN {X 0,Y 151.169,Z 538.282,A -85,B 0,C 180,E1 -24339.817,E2 -24339.817} C_VEL
LIN {X 0,Y 148.472,Z 541.714,A -85,B 0,C 180,E1 -24342.803,E2 -24342.803} C_VEL
LIN {X 0,Y 145.175,Z 545.448,A -85,B 0,C 180,E1 -24347.332,E2 -24347.332} C_VEL
LIN {X 0,Y 142.732,Z 547.923,A -85,B 0,C 180,E1 -24351.984,E2 -24351.984} C_VEL
LIN {X 0,Y 140.821,Z 549.389,A -85,B 0,C 180,E1 -24358.042,E2 -24358.042} C_VEL
LIN {X 0,Y 140.402,Z 549.589,A -85,B 0,C 180,E1 -24359.963,E2 -24359.963} C_VEL
LIN {X 0,Y 139.939,Z 549.1,A -85,B 0,C 180,E1 -24364.689,E2 -24364.689} C_VEL
LIN {X 0,Y 140.03,Z 547.531,A -85,B 0,C 180,E1 -24369.432,E2 -24369.432} C_VEL
LIN {X 0,Y 140.8,Z 544.89,A -85,B 0,C 180,E1 -24374.066,E2 -24374.066} C_VEL
LIN {X 0,Y 141.985,Z 541.143,A -85,B 0,C 180,E1 -24378.581,E2 -24378.581} C_VEL
LIN {X 0,Y 144.056,Z 535.168,A -85,B 0,C 180,E1 -24383.698,E2 -24383.698} C_VEL
LIN {X 0,Y 146.065,Z 529.838,A -85,B 0,C 180,E1 -24387.242,E2 -24387.242} C_VEL
LIN {X 0,Y 148.602,Z 523.364,A -85,B 0,C 180,E1 -24390.678,E2 -24390.678} C_VEL
LIN {X 0,Y 151.532,Z 515.531,A -85,B 0,C 180,E1 -24393.99,E2 -24393.99} C_VEL
LIN {X 0,Y 154.192,Z 508.093,A -85,B 0,C 180,E1 -24396.543,E2 -24396.543} C_VEL
LIN {X 0,Y 156.994,Z 499.904,A -85,B 0,C 180,E1 -24398.826,E2 -24398.826} C_VEL
LIN {X 0,Y 160.035,Z 489.751,A -85,B 0,C 180,E1 -24401.077,E2 -24401.077} C_VEL
LIN {X 0,Y 162.55,Z 479.951,A -85,B 0,C 180,E1 -24402.802,E2 -24402.802} C_VEL
LIN {X 0,Y 164.768,Z 469.765,A -85,B 0,C 180,E1 -24404.197,E2 -24404.197} C_VEL
LIN {X 0,Y 166.593,Z 458.68,A -85,B 0,C 180,E1 -24405.351,E2 -24405.351} C_VEL
LIN {X 0,Y 168.059,Z 447.905,A -85,B 0,C 180,E1 -24406.108,E2 -24406.108} C_VEL
